// Calls CyclicLogic of every registered CoE transfer and drops the ones that finished.
METHOD PRIVATE ServiceCoeTransfers
VAR
	i : UINT;
END_VAR
i := 0;
WHILE i < ActiveCoeCount DO
	ActiveCoe[i].CyclicLogic();
	IF ActiveCoe[i].Busy THEN
		i := i + 1;
	ELSE
		(* finished: move the last entry into the gap and service it in this cycle as well *)
		ActiveCoeCount			  := ActiveCoeCount - 1;
		ActiveCoe[i]			  := ActiveCoe[ActiveCoeCount];
		ActiveCoe[ActiveCoeCount] := 0;
	END_IF
END_WHILE
END_METHOD

METHOD PROTECTED SetError
VAR_INPUT
	Source	: E_EcErrorSource;
	ErrorId : UDINT;
END_VAR
_Error		 := TRUE;
_ErrorSource := Source;
_ErrorId	 := ErrorId;
END_METHOD

{attribute 'monitoring' := 'call'}
PROPERTY Simulated : BOOL
GET
Simulated := _Simulated;
END_GET
SET
_Simulated := Simulated;
END_SET
END_PROPERTY

{attribute 'monitoring' := 'call'}
PROPERTY SlaveCount : UINT
GET
SlaveCount := EcMaster.SlaveCount;
END_GET
END_PROPERTY

// TRUE if the slave is not in OP with a clean link (any state or link bit set).
METHOD PROTECTED SlaveNeedsDiagnostic : BOOL
VAR_INPUT
	Index : UINT;
END_VAR
SlaveNeedsDiagnostic := (SlavesState[Index].deviceState <> EC_DEVICE_STATE_OP) OR (SlavesState[Index].linkState <> 0);
END_METHOD

// Slave diagnostic sequence, run on every trigger (ChangeCount, slave count, frame WC state):
//  10/11 read all slave states (sized to the configured count)
//  12    classify, SLAVES_PER_CYCLE slaves per cycle; a clean network ends here
//  20/21 read the topology (hot connect flags) - only when a slave needs a diagnostic
//  30    evaluate from the first suspicious slave, stop at the first fault
//  40    assign the sync unit of every slave, once, after the sync units resolved their lists
METHOD PROTECTED SlaveState : BOOL
VAR
	k	: UINT;
	Idx : DINT;
END_VAR
GetSlaveTopologyInfo(sNetId	  := _MasterAmsNetId,
					 pAddrBuf := ADR(SlaveTopologyInfo),
					 cbBufLen := TopologyBufLen(),
					 tTimeout := ADS_TIMEOUT);

GetAllSlaveStates(sNetId	:= _MasterAmsNetId,
				  pStateBuf := ADR(SlavesState),
				  cbBufLen	:= SlaveCountUsed * SIZEOF(SlavesState[0]),
				  tTimeout	:= ADS_TIMEOUT);

CASE SlaveSequence OF
	(* Wait for a trigger *)
	0:
		IF RunSlaveDiag THEN
			RunSlaveDiag  := FALSE;
			SlaveSequence := 10;
		ELSIF NOT SyncUnitsAssigned AND_THEN SyncUnitsResolved() THEN
			EndDiagnosticPass();
		END_IF

	(* Read slave states *)
	10:
		GetAllSlaveStates.bExecute := TRUE;
		WaitCycles				   := 0;
		NextMinorStep(SlaveSequence);

	11:
		IF GetAllSlaveStates.bBusy THEN
			IF AdsWatchdogExpired(ADS_WAIT_CYCLES) THEN
				GetAllSlaveStates.bExecute := FALSE;
				FailSequence(E_EcErrorSource.Ads, ERROR_ADS_TIMEOUT);
			END_IF
		ELSIF GetAllSlaveStates.bError THEN
			GetAllSlaveStates.bExecute := FALSE;
			FailSequence(E_EcErrorSource.Ads, GetAllSlaveStates.nErrId);
		ELSE
			GetAllSlaveStates.bExecute := FALSE;
			ScanIndex				   := 0;
			AnyDiag					   := FALSE;
			FirstDiagIndex			   := 0;
			NextMinorStep(SlaveSequence);
		END_IF

	(* Classify: find the first slave that needs a diagnostic *)
	12:
		FOR k := 1 TO SLAVES_PER_CYCLE DO
			IF ScanIndex >= SlaveCountUsed THEN
				EXIT;
			END_IF

			IF SlaveNeedsDiagnostic(ScanIndex) THEN
				AnyDiag		   := TRUE;
				FirstDiagIndex := ScanIndex;
				EXIT;
			END_IF

			ScanIndex := ScanIndex + 1;
		END_FOR

		IF AnyDiag THEN
			SlaveSequence := 20;
		ELSIF ScanIndex >= SlaveCountUsed THEN
			EndDiagnosticPass(); // every slave OP with a clean link: no topology read, no evaluation
		END_IF

	(* Update topology *)
	20:
		GetSlaveTopologyInfo.bExecute := TRUE;
		WaitCycles					  := 0;
		NextMinorStep(SlaveSequence);

	21:
		IF GetSlaveTopologyInfo.bBusy THEN
			IF AdsWatchdogExpired(ADS_WAIT_CYCLES) THEN
				GetSlaveTopologyInfo.bExecute := FALSE;
				FailSequence(E_EcErrorSource.Ads, ERROR_ADS_TIMEOUT);
			END_IF
		ELSIF GetSlaveTopologyInfo.bError THEN
			GetSlaveTopologyInfo.bExecute := FALSE;
			FailSequence(E_EcErrorSource.Ads, GetSlaveTopologyInfo.nErrId);
		ELSE
			GetSlaveTopologyInfo.bExecute := FALSE;
			ScanIndex					  := FirstDiagIndex;
			SlaveSequence				  := 30;
		END_IF

	(* Evaluate slave errors from the first suspicious slave on *)
	30:
		FOR k := 1 TO SLAVES_PER_CYCLE DO
			IF ScanIndex >= SlaveCountUsed THEN
				EXIT;
			END_IF

			IF EvaluateSlave(ScanIndex) THEN
				ScanIndex := SlaveCountUsed; // fault latched: stop the pass
				EXIT;
			END_IF

			ScanIndex := ScanIndex + 1;
		END_FOR

		IF ScanIndex >= SlaveCountUsed THEN
			EndDiagnosticPass();
		END_IF

	(* Assign the sync unit of every slave (once) *)
	40:
		FOR k := 1 TO SLAVES_PER_CYCLE DO
			IF SyncUnitScan >= SYNC_UNITS THEN
				EXIT;
			END_IF

			IF ScanIndex >= SyncUnit[SyncUnitScan].SlaveCount THEN
				SyncUnitScan := SyncUnitScan + 1;
				ScanIndex	 := 0;
			ELSE
				Idx := GetSlaveIndexByAddr(SyncUnit[SyncUnitScan].SlaveAddress(ScanIndex));
				IF Idx >= 0 THEN
					IoDevice[Idx].SyncUnit := SyncUnit[SyncUnitScan];
				END_IF

				ScanIndex := ScanIndex + 1;
			END_IF
		END_FOR

		IF SyncUnitScan >= SYNC_UNITS THEN
			SyncUnitsAssigned := TRUE;
			SlaveSequence	  := 0;
		END_IF

ELSE
	(* Sequence error: unknown step *)
	FailSequence(E_EcErrorSource.Sequence, SlaveSequence);
END_CASE
END_METHOD

// TRUE once every sync unit has read and resolved its slave list.
METHOD PRIVATE SyncUnitsResolved : BOOL
VAR
	i : UINT;
END_VAR
SyncUnitsResolved := TRUE;
FOR i := 0 TO (SYNC_UNITS - 1) DO
	IF NOT SyncUnit[i].SlavesResolved THEN
		SyncUnitsResolved := FALSE;
		RETURN;
	END_IF
END_FOR
END_METHOD

// Byte length of the topology read: one entry per configured slave, not the whole array.
METHOD PRIVATE TopologyBufLen : UDINT
TopologyBufLen := SlaveCountUsed * SIZEOF(SlaveTopologyInfo[0]);
END_METHOD

END_FUNCTION_BLOCK

// ---- Component/CyclicComponent.TcPOU
FUNCTION_BLOCK ABSTRACT CyclicComponent EXTENDS Component IMPLEMENTS I_Cyclic
VAR
	RegisteredAsCyclicResult : RegistrationResult;
END_VAR

METHOD ABSTRACT CyclicLogic
END_METHOD

METHOD DeregisterWithParent
VAR_INPUT
	Parent : I_ContainComponents;
END_VAR
Parent.DeregisterComponent(THIS^);
Parent.DeregisterCyclic(THIS^);
END_METHOD

METHOD RegisterWithParent
VAR_INPUT
	Parent : I_ContainComponents;
END_VAR
RegisteredAsComponentResult := Parent.RegisterComponent(THIS^);
RegisteredAsCyclicResult := Parent.RegisterCyclic(THIS^);
END_METHOD

END_FUNCTION_BLOCK

// ---- Component/Component.TcPOU
FUNCTION_BLOCK ABSTRACT Component IMPLEMENTS I_Component
VAR
	_Name : T_MaxString;
	RegisteredAsComponentResult : RegistrationResult;
END_VAR

METHOD Accept
VAR_INPUT
	ComponentVisitor : I_ComponentVisitor;
END_VAR
ComponentVisitor.VisitComponent(THIS^);
END_METHOD

METHOD DeregisterWithParent
VAR_INPUT
	Parent : I_ContainComponents;
END_VAR
Parent.DeregisterComponent(THIS^);
END_METHOD

//FB_Init is always available implicitly and it is used primarily for initialization.

//The return value is not evaluated. For a specific influence, you can also declare the

//methods explicitly and provide additional code there with the standard initialization

//code. You can evaluate the return value.
METHOD FB_Init : BOOL
VAR_INPUT
	bInitRetains : BOOL; // TRUE: the retain variables are initialized (reset warm / reset cold)
	bInCopyCode	 : BOOL; // TRUE: the instance will be copied to the copy code afterward (online change)   
	Name		 : T_MaxString;
END_VAR
_Name := Name;
END_METHOD

{attribute 'monitoring' := 'call'}
PROPERTY Name : T_MaxString
GET
Name := _Name;
END_GET
SET
_Name := Name;
END_SET
END_PROPERTY

METHOD RegisterWithParent
VAR_INPUT
	Parent : I_ContainComponents;
END_VAR
RegisteredAsComponentResult := Parent.RegisterComponent(THIS^);
END_METHOD

END_FUNCTION_BLOCK

// ---- Components/EtherCat/SyncUnitTask.TcPOU
{attribute 'no_explicit_call' := 'do not call this POU directly'}
FUNCTION_BLOCK FINAL SyncUnitTask EXTENDS CyclicComponent IMPLEMENTS I_SyncUnitTask, I_Initializable, I_TaskResult, I_Simulatable
VAR
	SyncUnitTaskInfo AT %I* : ST_EtherCatSyncUnitTaskInfo;
	_SlaveCount				: UINT;
	_IsHotConnect			: BOOL;
	_SlavesResolved			: BOOL;
	// Resolves sync unit slave addresses to configured slaves (implemented by EtherCatMaster)
	Registry				: I_EcSlaveRegistry;
	SyncUnitSlaveAddresses	: ARRAY[0..MAX_EC_SLAVES] OF UINT;
	// TRUE at the configured slave index of every slave in this sync unit (filled by the resolve pass)
	MemberByIndex			: ARRAY[0..MAX_EC_SLAVES] OF BOOL;
END_VAR

VAR
	{attribute 'hide'}
	_Initialized : BOOL;
	{attribute 'hide'}
	_Error : BOOL;
	{attribute 'hide'}
	_Busy : BOOL;
	{attribute 'hide'}
	_ErrorId : UDINT;
	{attribute 'hide'}
	_Simulated : BOOL;
END_VAR

VAR
	SyncUnitState			  : UDINT := READ_SLAVES;
	ScanIndex				  : UINT;  // position of the multi-cycle resolve pass
	WaitCycles				  : UDINT; // ADS watchdog and retry delay
	ReadErrorLogged			  : BOOL;
	SlaveMessagePartA		  : STRING;
	SlaveMessagePartB		  : STRING;
	_EventProvider			  : I_EtherCatDiagnosticEventProvider;
	EcGetAllSyncUnitSlaveAddr : FB_EcGetAllSyncUnitSlaveAddr;
END_VAR

VAR CONSTANT
	ERROR_READ_SLAVE_NAMES	   : UDINT := 1;
	ERROR_REGISTER_SYNC_UNIT   : UDINT := 2;
	ERROR_VALID_DATA_SYNC_UNIT : UDINT := 3;
	STRING_LEN				   : INT   := 80;
	SYNC_UNIT_ALARM_MAX		   : UINT  := 3;

	//
	READ_SLAVES			  : UDINT := 0;
	READ_SLAVES_DONE	  : UDINT := 1;
	SYNC_UNIT_OK		  : UDINT := 2;
	RESOLVE_SLAVES		  : UDINT := 3;
	WORKING_COUNTER_ERROR : UDINT := 4;
	READ_ERROR			  : UDINT := 5;
	READ_RETRY_WAIT		  : UDINT := 6;
END_VAR

// Appends the name to the two event message parts while they have room (STRING_LEN each).
METHOD PRIVATE AppendSlaveName
VAR_INPUT
	SlaveName : STRING;
END_VAR

VAR
	Entry : STRING;
END_VAR
IF LEN(SlaveName) = 0 THEN
	RETURN;
END_IF

Entry := CONCAT(SlaveName, ', ');
IF (LEN(Entry) + LEN(SlaveMessagePartA)) <= STRING_LEN THEN
	SlaveMessagePartA := CONCAT(SlaveMessagePartA, Entry);
ELSIF (LEN(Entry) + LEN(SlaveMessagePartB)) <= STRING_LEN THEN
	SlaveMessagePartB := CONCAT(SlaveMessagePartB, Entry);
END_IF
END_METHOD

{attribute 'monitoring' := 'call'}
PROPERTY Busy : BOOL
GET
Busy := _Busy;
END_GET
END_PROPERTY

METHOD PUBLIC CyclicLogic
VAR
	k	 : UINT;
	Addr : UINT;
	Idx	 : DINT;
END_VAR
IF NOT Initialized THEN
	Initialize();
	RETURN;
END_IF

IF Simulated THEN
	RETURN;
END_IF

(* The slave list of a sync unit is configuration data: it is read once (retried on failure) and
   never re-read on working counter recovery. The buffer is sized to the configured slave count. *)
EcGetAllSyncUnitSlaveAddr(sNetId	:= '',
						  nObjectId := SyncUnitTaskInfo.ObjectId,
						  pAddrBuf	:= ADR(SyncUnitSlaveAddresses),
						  cbBufLen	:= SIZEOF(UINT) * MIN(Registry.ConfiguredSlaveCount, MAX_EC_SLAVES + 1),
						  tTimeout	:= T#5S);

EcGetAllSyncUnitSlaveAddr.bExecute := FALSE;
CASE SyncUnitState OF
	READ_SLAVES:
		EcGetAllSyncUnitSlaveAddr.bExecute := TRUE;
		WaitCycles						   := 0;
		SyncUnitState					   := READ_SLAVES_DONE;

	READ_SLAVES_DONE:
		IF EcGetAllSyncUnitSlaveAddr.bBusy THEN
			WaitCycles := WaitCycles + 1;
			IF WaitCycles > ADS_WAIT_CYCLES THEN
				SyncUnitState := READ_ERROR;
			END_IF
		ELSIF EcGetAllSyncUnitSlaveAddr.bError THEN
			SyncUnitState := READ_ERROR;
		ELSE
			_SlaveCount		  := EcGetAllSyncUnitSlaveAddr.nSlaves;
			ScanIndex		  := 0;
			_IsHotConnect	  := FALSE;
			SlaveMessagePartA := '';
			SlaveMessagePartB := '';
			MEMSET(ADR(MemberByIndex), 0, SIZEOF(MemberByIndex));
			SyncUnitState	  := RESOLVE_SLAVES;
		END_IF

	RESOLVE_SLAVES:
		(* Map every address to its configured slave through the slave registry of the master:
		   O(n) in total, SLAVES_PER_CYCLE slaves per cycle. *)
		FOR k := 1 TO SLAVES_PER_CYCLE DO
			IF ScanIndex >= _SlaveCount THEN
				EXIT;
			END_IF

			Addr := SyncUnitSlaveAddresses[ScanIndex];
			IF Addr <> 0 THEN
				Idx := Registry.GetSlaveIndexByAddr(Addr);
				IF Idx >= 0 THEN
					MemberByIndex[Idx] := TRUE;
					_IsHotConnect	   := _IsHotConnect OR Registry.IsHotConnectMember(DINT_TO_UINT(Idx));
					AppendSlaveName(Registry.GetSlaveName(DINT_TO_UINT(Idx)));
				END_IF
			END_IF

			ScanIndex := ScanIndex + 1;
		END_FOR

		IF ScanIndex >= _SlaveCount THEN
			_SlavesResolved := TRUE;
			SyncUnitState	:= SYNC_UNIT_OK;
		END_IF

	SYNC_UNIT_OK:
		IF SyncUnitTaskInfo.WcState THEN
			SyncUnitState := WORKING_COUNTER_ERROR;
			_Busy		  := TRUE;
		ELSE
			_Error	 := FALSE;
			_ErrorID := 0;
			_Busy	 := FALSE;
		END_IF

	WORKING_COUNTER_ERROR:
		_Busy	 := FALSE;
		_Error	 := TRUE;
		_ErrorID := ERROR_VALID_DATA_SYNC_UNIT;
		IF _EventProvider <> 0 THEN
			IF _IsHotConnect THEN
				_EventProvider.RaiseSyncUnitEvent(E_SyncUnit.SyncUnitWarning,
												  _Name,
												  SlaveMessagePartA,
												  SlaveMessagePartB);
			ELSE
				_EventProvider.RaiseSyncUnitEvent(E_SyncUnit.SyncUnitError,
												  _Name,
												  SlaveMessagePartA,
												  SlaveMessagePartB);
			END_IF
		END_IF

		IF NOT SyncUnitTaskInfo.WcState THEN
			IF _EventProvider <> 0 THEN
				_EventProvider.Reset();
			END_IF

			SyncUnitState := SYNC_UNIT_OK; // membership does not change on WC recovery: no re-read
		END_IF

	READ_ERROR:
		IF NOT ReadErrorLogged THEN
			Trace.LogMessage(Name, CONCAT('Sync Unit slave addresses could not be read! Error ID: ', TO_STRING(EcGetAllSyncUnitSlaveAddr.nErrId)));
			ReadErrorLogged := TRUE;
		END_IF

		_Error		  := TRUE;
		_ErrorID	  := ERROR_READ_SLAVE_NAMES;
		WaitCycles	  := 0;
		SyncUnitState := READ_RETRY_WAIT;

	READ_RETRY_WAIT:
		WaitCycles := WaitCycles + 1;
		IF WaitCycles > ADS_WAIT_CYCLES THEN
			SyncUnitState := READ_SLAVES;
		END_IF
END_CASE
END_METHOD

{attribute 'monitoring' := 'call'}
PROPERTY Error : BOOL
GET
Error := _Error;
END_GET
END_PROPERTY

{attribute 'monitoring' := 'call'}
PROPERTY ErrorId : UDINT
GET
ErrorId := _ErrorId;
END_GET
END_PROPERTY

PROPERTY EventProvider : I_EtherCatDiagnosticEventProvider
SET
_EventProvider := EventProvider;
END_SET
END_PROPERTY

(*FB_Init is always available implicitly and it is used primarily for initialization.
The return value is not evaluated. For a specific influence, you can also declare the
methods explicitly and provide additional code there with the standard initialization
code. You can evaluate the return value.*)
METHOD FB_Init : BOOL
VAR_INPUT
	(* TRUE: the retain variables are initialized (reset warm / reset cold)*)
	bInitRetains : BOOL;

	(* TRUE: the instance will be copied to the copy code afterward (online change)   *)
	bInCopyCode			: BOOL;
	Name	 : T_MaxString;
	Registry : I_EcSlaveRegistry;
END_VAR
THIS^.Registry := Registry;
END_METHOD

METHOD Initialize
VAR_INPUT
END_VAR
IF NOT _Error AND NOT Simulated AND F_GetMappingStatus(ADR(SyncUnitTaskInfo.ObjectId), SIZEOF(SyncUnitTaskInfo.ObjectId)) = EplcMappingStatus.MS_Unmapped THEN
	_Error := TRUE;
	Trace.LogMessage(Name, 'Init Failed - SyncUnitTaskInfo.ObjectId not mapped to the sync unit diagnostic!');
END_IF

IF NOT _Error AND NOT Simulated AND F_GetMappingStatus(ADR(SyncUnitTaskInfo.SlaveCount), SIZEOF(SyncUnitTaskInfo.SlaveCount)) = EplcMappingStatus.MS_Unmapped THEN
	_Error := TRUE;
	Trace.LogMessage(Name, 'Init Failed - SyncUnitTaskInfo.SlaveCount not mapped to the sync unit diagnostic!');
END_IF

IF NOT _Error AND NOT Simulated AND F_GetMappingStatus(ADR(SyncUnitTaskInfo.State), SIZEOF(SyncUnitTaskInfo.State)) = EplcMappingStatus.MS_Unmapped THEN
	_Error := TRUE;
	Trace.LogMessage(Name, 'Init Failed - SyncUnitTaskInfo.State not mapped to the sync unit diagnostic!');
END_IF

IF NOT _Error AND NOT Simulated AND F_GetMappingStatus(ADR(SyncUnitTaskInfo.WcState), SIZEOF(SyncUnitTaskInfo.WcState)) = EplcMappingStatus.MS_Unmapped THEN
	_Error := TRUE;
	Trace.LogMessage(Name, 'Init Failed - SyncUnitTaskInfo.WcState not mapped to the sync unit diagnostic!');
END_IF

IF _Error THEN
	RETURN;
END_IF

IF Simulated THEN
	_Initialized := TRUE;
	RETURN;
END_IF

F_EcGetSyncUnitName(SyncUnitTaskInfo.ObjectId, sSyncUnitName => _Name);
_Initialized := TRUE;
END_METHOD

{attribute 'monitoring' := 'call'}
PROPERTY Initialized : BOOL
GET
Initialized := _Initialized;
END_GET
SET
_Initialized := Initialized;
END_SET
END_PROPERTY

{attribute 'monitoring' := 'call'}
PROPERTY IoDataValid : BOOL
GET
IoDataValid := NOT SyncUnitTaskInfo.WcState;
END_GET
END_PROPERTY

// TRUE if at least one slave of this sync unit belongs to a hot connect group.
{attribute 'monitoring' := 'call'}
PROPERTY IsHotConnect : BOOL
GET
IsHotConnect := _IsHotConnect;
END_GET
END_PROPERTY

// O(1) once the slave list is resolved (SlavesResolved).
METHOD IsTerminalPartOfSyncUnit : BOOL
VAR_INPUT
	Addr : UINT;
END_VAR

VAR
	Idx : DINT;
END_VAR
Idx						 := Registry.GetSlaveIndexByAddr(Addr);
IsTerminalPartOfSyncUnit := (Idx >= 0) AND_THEN MemberByIndex[Idx];
END_METHOD

{attribute 'monitoring' := 'call'}
PROPERTY Simulated : BOOL
GET
Simulated := _Simulated;
END_GET
SET
_Simulated := Simulated;
END_SET
END_PROPERTY

// EtherCAT address of the slave at Position (0..SlaveCount-1) in this sync unit; 0 if out of range.
METHOD SlaveAddress : UINT
VAR_INPUT
	Position : UINT;
END_VAR
IF Position < _SlaveCount THEN
	SlaveAddress := SyncUnitSlaveAddresses[Position];
END_IF
END_METHOD

{attribute 'monitoring' := 'call'}
PROPERTY PUBLIC SlaveCount : UINT
GET
SlaveCount := _SlaveCount;
END_GET
END_PROPERTY

// TRUE once the slave list has been read and mapped to the configured slaves.
{attribute 'monitoring' := 'call'}
PROPERTY SlavesResolved : BOOL
GET
SlavesResolved := _SlavesResolved;
END_GET
END_PROPERTY

END_FUNCTION_BLOCK

// ---- Tracing/Trace.TcPOU
FUNCTION_BLOCK Trace
VAR_GENERIC CONSTANT
	MaxCount : UDINT := 10;
END_VAR IMPLEMENTS I_TracePublisher, I_Trace, I_TraceLogger
VAR
	Loggers : ARRAY[0..MaxCount] OF I_TraceLogger;
	_TraceLevel : TcEventSeverityExt := TcEventSeverityExt.Warning;
END_VAR

METHOD Critical
VAR_INPUT
	Source	  : T_MaxString;
	Message	  : T_MaxString;
END_VAR
VAR
	i : UDINT;
END_VAR
FOR i := 0 TO MaxCount DO
	IF Loggers[i] <> 0 AND_THEN _TraceLevel < 5 THEN
		Loggers[i].LogMessage(Source,
							  Message,
							  0,
							  0,
							  1,
							  4);
	END_IF
END_FOR
END_METHOD

METHOD Error
VAR_INPUT
	Source	  : T_MaxString;
	Message	  : T_MaxString;
END_VAR
VAR
	i : UDINT;
END_VAR
FOR i := 0 TO MaxCount DO
	IF Loggers[i] <> 0 AND_THEN _TraceLevel < 4 THEN
		Loggers[i].LogMessage(Source,
							  Message,
							  0,
							  0,
							  1,
							  3);
	END_IF
END_FOR
END_METHOD

METHOD Info
VAR_INPUT
	Source	  : T_MaxString;
	Message	  : T_MaxString;
END_VAR
VAR
	i : UDINT;
END_VAR
FOR i := 0 TO MaxCount DO
	IF Loggers[i] <> 0 AND_THEN _TraceLevel < 2 THEN
		Loggers[i].LogMessage(Source,
							  Message,
							  0,
							  0,
							  1,
							  1);
	END_IF
END_FOR
END_METHOD

METHOD LogMessage
VAR_INPUT
	Key		  : T_MaxString;
	Value	  : T_MaxString;
	SourceId  : UDINT := 0;
	TimeStamp : ULINT := 0;
	MessageId : UDINT := 1;
	Severity  : USINT := 1;
END_VAR

VAR
	i : UDINT;
END_VAR
FOR i := 0 TO MaxCount DO
	IF Loggers[i] <> 0 THEN
		Loggers[i].LogMessage(Key,
							  Value,
							  SourceId,
							  TimeStamp,
							  MessageId,
							  Severity);
	END_IF
END_FOR
END_METHOD

METHOD Subscribe
VAR_INPUT
	Logger : I_TraceLogger;
END_VAR

VAR
	i : UDINT;
END_VAR
FOR i := 0 TO ApplicationBaseParameter.MaxCountInCollections DO
	IF Loggers[i] = 0 THEN
		Loggers[i] := Logger;
		EXIT;
	END_IF
END_FOR
END_METHOD

PROPERTY TraceLevel : TcEventSeverityExt
GET
TraceLevel := _TraceLevel;
END_GET
SET
_TraceLevel := TraceLevel;
END_SET
END_PROPERTY

METHOD Unsubscribe
VAR_INPUT
	Logger : I_TraceLogger;
END_VAR

VAR
	i : UDINT;
END_VAR
FOR i := 0 TO ApplicationBaseParameter.MaxCountInCollections DO
	IF Loggers[i] = Logger THEN
		Loggers[i] := 0;
		EXIT;
	END_IF
END_FOR
END_METHOD

METHOD Verbose
VAR_INPUT
	Source	  : T_MaxString;
	Message	  : T_MaxString;
END_VAR
VAR
	i : UDINT;
END_VAR
FOR i := 0 TO MaxCount DO
	IF Loggers[i] <> 0 AND_THEN _TraceLevel = 0 THEN
		Loggers[i].LogMessage(Source,
							  Message,
							  0,
							  0,
							  1,
							  0);
	END_IF
END_FOR
END_METHOD

METHOD Warning
VAR_INPUT
	Source	  : T_MaxString;
	Message	  : T_MaxString;
END_VAR
VAR
	i : UDINT;
END_VAR
FOR i := 0 TO MaxCount DO
	IF Loggers[i] <> 0 AND_THEN _TraceLevel < 3 THEN
		Loggers[i].LogMessage(Source,
							  Message,
							  0,
							  0,
							  1,
							  2);
	END_IF
END_FOR
END_METHOD

END_FUNCTION_BLOCK

// ---- Statemachine/Generic/State.TcPOU
FUNCTION_BLOCK ABSTRACT State IMPLEMENTS I_State
VAR
	Statemachine  : I_Statemachine;
	SequenceState : UDINT;
END_VAR

METHOD Executing : BOOL
Executing := TRUE;
END_METHOD

//FB_Init is always available implicitly and it is used primarily for initialization.

//The return value is not evaluated. For a specific influence, you can also declare the

//methods explicitly and provide additional code there with the standard initialization

//code. You can evaluate the return value.
METHOD FB_Init : BOOL
VAR_INPUT
	bInitRetains : BOOL; // TRUE: the retain variables are initialized (reset warm / reset cold)
	bInCopyCode	 : BOOL; // TRUE: the instance will be copied to the copy code afterward (online change)  
	State		 : DINT;
	Statemachine : I_Statemachine;
END_VAR
THIS^.Statemachine := Statemachine;
IF THIS^.Statemachine <> 0 THEN
	THIS^.Statemachine.States.AddStateAtIndex(State, THIS^);
END_IF
END_METHOD

METHOD Inactive
SequenceState := 0;
END_METHOD

END_FUNCTION_BLOCK

// ---- Statemachine/Generic/Statemachine.TcPOU
FUNCTION_BLOCK Statemachine
VAR_GENERIC CONSTANT
	InitialState : DINT := 1;
END_VAR
EXTENDS CyclicComponent IMPLEMENTS I_Statemachine
VAR
	StateList	  : StateList<TO_DINT(ApplicationBaseParameter.MaxCountInCollections)>;
	_CurrentState : DINT := InitialState;
	{attribute 'hide'}
	DefaultModeController : ModeControl;
	_Mode				  : I_Mode := DefaultModeController;
END_VAR

METHOD ChangeState
VAR_INPUT
	StateCommand : DINT;
END_VAR
IF StateList.NumberOfStates = 0 THEN
	Trace.LogMessage('Statemachine', 'No states defined!');
	RETURN;
END_IF

_CurrentState := StateCommand;
END_METHOD

{attribute 'monitoring' := 'call'}
PROPERTY CurrentState : DINT
GET
CurrentState := _CurrentState;
END_GET
END_PROPERTY

METHOD CyclicLogic
VAR
	i	  : DINT;
	State : I_State;
END_VAR
IF StateList.NumberOfStates = 0 THEN
	RETURN;
END_IF

FOR i := 0 TO (StateList.NumberOfStates - 1) DO
	State := StateList.GetStateAtIndex(i);
	IF State <> 0 THEN
		IF (i = _CurrentState) THEN
			State.Executing();
		ELSE
			State.Inactive();
		END_IF
	END_IF
END_FOR
END_METHOD

PROPERTY Mode : I_Mode
GET
Mode := _Mode;
END_GET
SET
_Mode := Mode;
END_SET
END_PROPERTY

PROPERTY States : I_StateList
GET
States := StateList;
END_GET
END_PROPERTY

END_FUNCTION_BLOCK

// ---- _Internal/Statemachine/StateList.TcPOU
FUNCTION_BLOCK StateList
VAR_GENERIC CONSTANT
	MaxCount : DINT := 10;
END_VAR IMPLEMENTS I_StateList
VAR
	States : ARRAY[0..MaxCount] OF I_State;
END_VAR

METHOD AddStateAtIndex
VAR_INPUT
	Index : DINT;
	State : I_State;
END_VAR
IF Index > MaxCount THEN
	RETURN;
END_IF

States[Index] := State;
END_METHOD

METHOD GetStateAtIndex : I_State
VAR_INPUT
	Index : DINT;
END_VAR
IF Index > MaxCount THEN
	RETURN;
END_IF

GetStateAtIndex := States[Index];
END_METHOD

PROPERTY NumberOfStates : DINT
GET
NumberOfStates := MaxCount;
END_GET
END_PROPERTY

END_FUNCTION_BLOCK

// ---- Modes/ModeControl.TcPOU
FUNCTION_BLOCK ModeControl IMPLEMENTS I_Mode
VAR
	{attribute 'hide'}
	_CurrentMode : DINT := 1;
END_VAR

METHOD ChangeMode
VAR_INPUT
	RequestedMode : DINT;
END_VAR
IF (RequestedMode >= 1) THEN
	_CurrentMode := RequestedMode;
ELSE
	Trace.LogMessage('Mode Controller', 'Requested Mode is not Defined');
END_IF
END_METHOD

{attribute 'monitoring' := 'call'}
PROPERTY CurrentMode : DINT
GET
CurrentMode := _CurrentMode;
END_GET
END_PROPERTY

END_FUNCTION_BLOCK

// ---- Components/EtherCat/EtherCatIoDevice.TcPOU
FUNCTION_BLOCK EtherCatIoDevice EXTENDS CyclicComponent IMPLEMENTS I_EcIoDevice
VAR
	_Config		  : REFERENCE TO ST_EcSlaveConfigData;
	_State		  : REFERENCE TO ST_EcExtendedSlaveState;
	_SyncUnit	  : I_SyncUnitTask;
	_CoeScheduler : I_CoeTransferScheduler;
	_AmsAddr	  : AMSADDR;
	CoeDevice	  : CoeDevice('CoE Terminal');
	{attribute 'hide'}
	NullCoeDevice : NullCoeDevice('Null Terminal');
END_VAR

PROPERTY AmsNetId : AMSNETID
SET
_AmsAddr.netId := AmsNetId;
END_SET
END_PROPERTY

{attribute 'monitoring' := 'call'}
PROPERTY Bootstrap : BOOL
GET
VAR
	DiagByte : BYTE;
END_VAR
IF __ISVALIDREF(_State) THEN
	DiagByte  := _State.deviceState AND 16#0F;
	Bootstrap := DiagByte = EC_DEVICE_STATE_BOOTSTRAP;
END_IF
END_GET
END_PROPERTY

// CoE access of this slave; NullCoeDevice when the slave has no mailbox (or no configuration yet).
PROPERTY CoE : I_CoeDevice
GET
IF NOT __ISVALIDREF(_Config) OR_ELSE _Config.nMailboxInSize = 0 THEN
	CoE := NullCoeDevice;
ELSE
	CoE := CoeDevice;
END_IF
END_GET
SET
END_SET
END_PROPERTY

// Scheduler that services this slave's CoE transfers (set by EtherCatMaster during Initialize).
// Without one, CyclicLogic must be called each cycle while CoE.Busy.
PROPERTY CoeScheduler : I_CoeTransferScheduler
SET
_CoeScheduler		:= CoeScheduler;
CoeDevice.Scheduler := CoeScheduler;
END_SET
END_PROPERTY

PROPERTY Configuration : REFERENCE TO ST_EcSlaveConfigData
GET
Configuration REF= _Config;
END_GET
SET
_Config REF= Configuration;

(* The CoE mailbox is addressed by the EtherCAT address of the slave. *)
IF __ISVALIDREF(_Config) THEN
	_AmsAddr.port	  := _Config.nAddr;
	CoeDevice.AdsAddr REF= _AmsAddr;
END_IF
END_SET
END_PROPERTY

// Services a CoE transfer in flight when no CoeScheduler is attached. With a scheduler
// (the normal case under EtherCatMaster) this method does nothing.
METHOD CyclicLogic
IF _CoeScheduler <> 0 THEN
	RETURN;
END_IF

IF __ISVALIDREF(_Config) AND_THEN _Config.nMailboxInSize <> 0 AND_THEN CoeDevice.Busy THEN
	CoeDevice.CyclicLogic();
END_IF
END_METHOD

// EC_DEVICE_STATE_ERROR: state machine error in the slave (deviceState bit 4).
{attribute 'monitoring' := 'call'}
PROPERTY DeviceError : BOOL
GET
IF __ISVALIDREF(_State) THEN
	DeviceError := _State.deviceState.4;
END_IF
END_GET
END_PROPERTY

// EC_DEVICE_STATE_DISABLED: slave is disabled in the configuration (deviceState bit 7).
{attribute 'monitoring' := 'call'}
PROPERTY Disabled : BOOL
GET
IF __ISVALIDREF(_State) THEN
	Disabled := _State.deviceState.7;
END_IF
END_GET
END_PROPERTY

{attribute 'monitoring' := 'call'}
PROPERTY Init : BOOL
GET
VAR
	DiagByte : BYTE;
END_VAR
IF __ISVALIDREF(_State) THEN
	DiagByte := _State.deviceState AND 16#0F;
	Init	 := DiagByte = EC_DEVICE_STATE_INIT;
END_IF
END_GET
END_PROPERTY

// EC_DEVICE_STATE_INITCMD_ERROR: error while sending the init commands (deviceState bit 6).
{attribute 'monitoring' := 'call'}
PROPERTY InitCmdError : BOOL
GET
IF __ISVALIDREF(_State) THEN
	InitCmdError := _State.deviceState.6;
END_IF
END_GET
END_PROPERTY

// EC_DEVICE_STATE_INVALID_VPRS: vendor id / product code / revision / serial mismatch (deviceState bit 5).
{attribute 'monitoring' := 'call'}
PROPERTY InvalidVPRS : BOOL
GET
IF __ISVALIDREF(_State) THEN
	InvalidVPRS := _State.deviceState.5;
END_IF
END_GET
END_PROPERTY

{attribute 'monitoring' := 'call'}
PROPERTY IoDataValid : BOOL
GET
IF _SyncUnit <> 0 THEN
	IoDataValid := _SyncUnit.IoDataValid;
ELSE
	IoDataValid := TRUE;
END_IF
END_GET
END_PROPERTY

{attribute 'monitoring' := 'call'}
PROPERTY OP : BOOL
GET
VAR
	DiagByte : BYTE;
END_VAR
IF __ISVALIDREF(_State) THEN
	DiagByte := _State.deviceState AND 16#0F;
	OP		 := DiagByte = EC_DEVICE_STATE_OP;
END_IF
END_GET
END_PROPERTY

{attribute 'monitoring' := 'call'}
PROPERTY PreOp : BOOL
GET
VAR
	DiagByte : BYTE;
END_VAR
IF __ISVALIDREF(_State) THEN
	DiagByte := _State.deviceState AND 16#0F;
	PreOp	 := DiagByte = EC_DEVICE_STATE_PREOP;
END_IF
END_GET
END_PROPERTY

{attribute 'monitoring' := 'call'}
PROPERTY SafeOp : BOOL
GET
VAR
	DiagByte : BYTE;
END_VAR
IF __ISVALIDREF(_State) THEN
	DiagByte := _State.deviceState AND 16#0F;
	SafeOp	 := DiagByte = EC_DEVICE_STATE_SAFEOP;
END_IF
END_GET
END_PROPERTY

PROPERTY State : REFERENCE TO ST_EcExtendedSlaveState
GET
State REF= _State;
END_GET
SET
_State REF= State;
END_SET
END_PROPERTY

PROPERTY SyncUnit : I_SyncUnitTask
SET
_SyncUnit := SyncUnit;
END_SET
END_PROPERTY

END_FUNCTION_BLOCK

// ---- Components/CoE/CoeDevice.TcPOU
FUNCTION_BLOCK CoeDevice EXTENDS CyclicComponent IMPLEMENTS I_CoeDevice, I_CoeTransfer
VAR
	{attribute 'hide'}
	_Error : BOOL;
	{attribute 'hide'}
	_Busy : BOOL;
	{attribute 'hide'}
	_ErrorId : UDINT;
	{attribute 'hide'}
	_ActiveIsWrite : BOOL;
	_AdsAddr   : REFERENCE TO AMSADDR;
	_Scheduler : I_CoeTransferScheduler; // optional: services this device while a transfer is in flight
	CoeRead	   : FB_EcCoESdoReadEx;
	CoeWrite   : FB_EcCoESdoWriteEx;
END_VAR

VAR CONSTANT
	ERROR_NO_ADDRESS : UDINT := 16#70B; // ADS: invalid parameter - AdsAddr reference not set
END_VAR

PROPERTY AdsAddr : REFERENCE TO AMSADDR
GET
AdsAddr REF= _AdsAddr;
END_GET
SET
_AdsAddr REF= AdsAddr;
END_SET
END_PROPERTY

{attribute 'monitoring' := 'call'}
PROPERTY Busy : BOOL
GET
Busy := _Busy;
END_GET
END_PROPERTY

// Services the SDO transfer in flight. Call each cycle while Busy; with a Scheduler set the
// scheduler does this for you.
METHOD CyclicLogic
VAR_INST
END_VAR
IF NOT __ISVALIDREF(_AdsAddr) THEN
	RETURN;
END_IF

CoeRead(sNetId := F_CreateAmsNetId(_AdsAddr.netId), nSlaveAddr := _AdsAddr.port, tTimeout := T#1S);
CoeWrite(sNetId := F_CreateAmsNetId(_AdsAddr.netId), nSlaveAddr := _AdsAddr.port, tTimeout := T#1S);
CoeRead.bExecute  := FALSE;
CoeWrite.bExecute := FALSE;

(* Only the active function block decides Busy/Error: a stale bError of the other one must not leak. *)
IF _ActiveIsWrite THEN
	_Busy := CoeWrite.bBusy;
	IF CoeWrite.bError THEN
		_Error	 := TRUE;
		_ErrorId := CoeWrite.nErrId;
	END_IF
ELSE
	_Busy := CoeRead.bBusy;
	IF CoeRead.bError THEN
		_Error	 := TRUE;
		_ErrorId := CoeRead.nErrId;
	END_IF
END_IF
END_METHOD

{attribute 'monitoring' := 'call'}
PROPERTY Error : BOOL
GET
Error := _Error;
END_GET
END_PROPERTY

{attribute 'monitoring' := 'call'}
PROPERTY ErrorId : UDINT
GET
ErrorID := _ErrorID;
END_GET
END_PROPERTY

// Starts an SDO read; ignored while Busy. Fails with ERROR_NO_ADDRESS if AdsAddr is not set.
METHOD Read
VAR_INPUT
	Index	 : WORD;
	SubIndex : BYTE;
	pDstBuf	 : PVOID;
	BufLen	 : UDINT;
END_VAR
IF _Busy THEN
	RETURN;
END_IF

IF NOT __ISVALIDREF(_AdsAddr) THEN
	_Error	 := TRUE;
	_ErrorId := ERROR_NO_ADDRESS;
	RETURN;
END_IF

CoeRead.nSubIndex		:= SubIndex;
CoeRead.nIndex			:= Index;
CoeRead.pDstBuf			:= pDstBuf;
CoeRead.cbBufLen		:= BufLen;
CoeRead.bCompleteAccess := SubIndex = 0;
_ActiveIsWrite			:= FALSE;
_Error					:= FALSE;
_ErrorId				:= 0;
_Busy					:= TRUE;
CoeRead.bExecute		:= TRUE;

IF _Scheduler <> 0 THEN
	_Scheduler.Register(THIS^);
END_IF
END_METHOD

// Optional scheduler that calls CyclicLogic while a transfer is in flight (set by EtherCatIoDevice).
PROPERTY Scheduler : I_CoeTransferScheduler
GET
Scheduler := _Scheduler;
END_GET
SET
_Scheduler := Scheduler;
END_SET
END_PROPERTY

// Starts an SDO write from pDstBuf (used as the source buffer); ignored while Busy.
METHOD Write
VAR_INPUT
	Index	 : WORD;
	SubIndex : BYTE;
	pDstBuf	 : PVOID;
	BufLen	 : UDINT;
END_VAR
IF _Busy THEN
	RETURN;
END_IF

IF NOT __ISVALIDREF(_AdsAddr) THEN
	_Error	 := TRUE;
	_ErrorId := ERROR_NO_ADDRESS;
	RETURN;
END_IF

CoeWrite.nSubIndex		 := SubIndex;
CoeWrite.nIndex			 := Index;
CoeWrite.pSrcBuf		 := pDstBuf;
CoeWrite.cbBufLen		 := BufLen;
CoeWrite.bCompleteAccess := SubIndex = 0;
_ActiveIsWrite			 := TRUE;
_Error					 := FALSE;
_ErrorId				 := 0;
_Busy					 := TRUE;
CoeWrite.bExecute		 := TRUE;

IF _Scheduler <> 0 THEN
	_Scheduler.Register(THIS^);
END_IF
END_METHOD

END_FUNCTION_BLOCK

// ---- Components/CoE/NullCoeDevice.TcPOU
FUNCTION_BLOCK NullCoeDevice EXTENDS CyclicComponent IMPLEMENTS I_CoeDevice
VAR
END_VAR

PROPERTY AdsAddr : REFERENCE TO AMSADDR
GET
END_GET
SET
END_SET
END_PROPERTY

{attribute 'monitoring' := 'call'}
PROPERTY Busy : BOOL
GET
END_GET
END_PROPERTY

METHOD CyclicLogic
END_METHOD

{attribute 'monitoring' := 'call'}
PROPERTY Error : BOOL
GET
END_GET
END_PROPERTY

{attribute 'monitoring' := 'call'}
PROPERTY ErrorId : UDINT
GET
END_GET
END_PROPERTY

METHOD Read
VAR_INPUT
	Index	 : WORD;
	SubIndex : BYTE;
	pDstBuf	 : PVOID;
	BufLen	 : UDINT;
END_VAR
END_METHOD

METHOD Write
VAR_INPUT
	Index	 : WORD;
	SubIndex : BYTE;
	pDstBuf	 : PVOID;
	BufLen	 : UDINT;
END_VAR
END_METHOD

END_FUNCTION_BLOCK

// ---- Motion/MC3/Mc3Axis.TcPOU
FUNCTION_BLOCK Mc3Axis EXTENDS CyclicComponent IMPLEMENTS I_Initializable, I_Mc3Axis
VAR
	_Axis				 : REFERENCE TO Tc3_Mc3Ptp.AXIS_REF;
	Defaults			 : ST_Mc3MotionDefaults;
	MotionTaskCollection : Mc3MotionTaskCollection<ApplicationBaseMotionParameter.MaxMotionTasks>(THIS^);

	// Tasks
	PowerTask  : Mc3PowerTask	 := (Name := 'MC Power');
	JogTask	   : Mc3MoveJogTask	 := (Name := 'MC Jog');
	_StopTask  : I_Mc3MotionTask := Defaults.DefaultStopTask;
	_ResetTask : I_Mc3MotionTask := Defaults.DefaultResetTask;
	_HomeTask  : I_Mc3MotionTask := Defaults.DefaultHomeTask;
	SetOverride : Tc3_Mc3Ptp.MC_SetOverride;

	// Initialization is delegated to its own component
	ParameterLoader : Mc3AxisParameterLoader<ApplicationBaseMotionParameter.MaxAxisParameters>;
	_Initialized		: BOOL;
	// TRUE once a parent module owns our Initialize() call
	{attribute 'hide'}
	_InitializeDrivenByParent : BOOL;
	{attribute 'hide'}
	_LoadErrorLogged		  : BOOL;

	//
	_Acceleration : LREAL;
	_Deceleration : LREAL;
	_Velocity	  : LREAL;
	_Jerk		  : LREAL;
	_McBufferMode : Tc3_Mc3Ptp.EBufferMode		:= Tc3_Mc3Ptp.EBufferMode.Aborting;
	_Direction	  : Tc3_Mc3Ptp.EModuloDirection := Tc3_Mc3Ptp.EModuloDirection.ShortestDistance;
	_JogMode	  : Tc3_Mc3Ptp.EJogMode			:= Tc3_Mc3Ptp.EJogMode.StandardSlow;
END_VAR

{attribute 'monitoring' := 'call'}
PROPERTY Acceleration : LREAL
GET
Acceleration := _Acceleration;
END_GET
SET
_Acceleration := Acceleration;
END_SET
END_PROPERTY

{attribute 'monitoring' := 'call'}
PROPERTY ActualAcceleration : LREAL
GET
ActualAcceleration := _Axis.McToPlc.Act.Acceleration;
END_GET
END_PROPERTY

{attribute 'monitoring' := 'call'}
PROPERTY ActualPosition : LREAL
GET
ActualPosition := _Axis.McToPlc.Act.Position;
END_GET
END_PROPERTY

{attribute 'monitoring' := 'call'}
PROPERTY ActualPositionModulo : LREAL
GET
ActualPositionModulo := _Axis.McToPlc.Modulo.ActPosition;
END_GET
END_PROPERTY

{attribute 'monitoring' := 'call'}
PROPERTY ActualTorque : LREAL
GET
ActualTorque := _Axis.McToPlc.Act.Torque;
END_GET
END_PROPERTY

{attribute 'monitoring' := 'call'}
PROPERTY ActualVelocity : LREAL
GET
ActualVelocity := _Axis.McToPlc.Act.Velocity;
END_GET
END_PROPERTY

PROPERTY Axis : REFERENCE TO Tc3_Mc3Ptp.AXIS_REF
GET
Axis REF= _Axis;
END_GET
END_PROPERTY

PROPERTY BufferMode : REFERENCE TO Tc3_Mc3Ptp.EBufferMode
GET
BufferMode REF= _McBufferMode;
END_GET
END_PROPERTY

{attribute 'monitoring' := 'call'}
PROPERTY Busy : BOOL
GET
Busy := MotionTaskCollection.Busy;
END_GET
END_PROPERTY

METHOD CyclicLogic
IF NOT _Initialized THEN
	// A parent module drives Initialize() through its Initializer. Only
	// self-initialize when there is no parent, so the call has one owner.
	IF NOT _InitializeDrivenByParent THEN
		Initialize();
	END_IF

	RETURN;
END_IF

MotionTaskCollection.CyclicLogic();
END_METHOD

{attribute 'monitoring' := 'call'}
PROPERTY Coupled : BOOL
GET
Coupled := _Axis.McToPlc.Std.AxisState = EAxisState.SynchronizedMotion;
END_GET
END_PROPERTY

{attribute 'monitoring' := 'call'}
PROPERTY Deceleration : LREAL
GET
Deceleration := _Deceleration;
END_GET
SET
_Deceleration := Deceleration;
END_SET
END_PROPERTY

PROPERTY Direction : REFERENCE TO Tc3_Mc3Ptp.EModuloDirection
GET
Direction REF= _Direction;
END_GET
END_PROPERTY

{attribute 'monitoring' := 'call'}
PROPERTY Disabled : BOOL
GET
Disabled := NOT PowerTask.Enabled;
END_GET
END_PROPERTY

METHOD Disable
PowerTask.Disable();
END_METHOD

METHOD Enable
IF Error THEN
	RETURN;
END_IF

PowerTask.Enable();
END_METHOD

{attribute 'monitoring' := 'call'}
PROPERTY Enabled : BOOL
GET
Enabled := PowerTask.Enabled;
END_GET
END_PROPERTY

{attribute 'monitoring' := 'call'}
PROPERTY Error : BOOL
GET
Error := MotionTaskCollection.Error OR (_Axis.McToPlc.Std.AxisState = EAxisState.ErrorStop);
END_GET
END_PROPERTY

{attribute 'monitoring' := 'call'}
PROPERTY ErrorId : UDINT
GET
IF _Axis.McToPlc.Std.ErrorId <> 0 THEN
	ErrorId := _Axis.McToPlc.Std.ErrorId;
	RETURN;
END_IF

ErrorId := MotionTaskCollection.ErrorId;
END_GET
END_PROPERTY

(*FB_Init is always available implicitly and it is used primarily for initialization.
The return value is not evaluated. For a specific influence, you can also declare the
methods explicitly and provide additional code there with the standard initialization
code. You can evaluate the return value.*)
METHOD FB_Init : BOOL
VAR_INPUT
	(* TRUE: the retain variables are initialized (reset warm / reset cold)*)
	bInitRetains : BOOL;

	(* TRUE: the instance will be copied to the copy code afterward (online change)   *)
	bInCopyCode : BOOL;
	Name		: T_MaxString;
	Axis		: REFERENCE TO Tc3_Mc3Ptp.AXIS_REF;
END_VAR
_Axis REF= Axis;

// Declare which NC parameters pre-load the dynamics properties.
// Adding one is a single line here - there is no sequence to edit.
ParameterLoader.Configure(_Axis);
ParameterLoader.AddParameter(EAxisParameterId.DefaultAcceleration, ADR(_Acceleration));
ParameterLoader.AddParameter(EAxisParameterId.DefaultDeceleration, ADR(_Deceleration));
ParameterLoader.AddParameter(EAxisParameterId.DefaultJerk, ADR(_Jerk));
ParameterLoader.AddParameter(EAxisParameterId.MaximumVelocity, ADR(_Velocity));

// Register all Motion Tasks to Collection
MotionTaskCollection.AddTask(PowerTask);
MotionTaskCollection.AddTask(_StopTask);
MotionTaskCollection.AddTask(_ResetTask);
MotionTaskCollection.AddTask(_HomeTask);
MotionTaskCollection.AddTask(JogTask);
END_METHOD

METHOD Home
VAR_INPUT
END_VAR
IF Coupled THEN
	// Homing a coupled axis is meaningless - decouple first
	RETURN;
END_IF

_HomeTask.Execute();
END_METHOD

PROPERTY HomeTask : I_Mc3MotionTask
SET
MotionTaskCollection.RemoveTaskByInstance(_HomeTask);
_HomeTask := HomeTask;
MotionTaskCollection.AddTask(_HomeTask);
END_SET
END_PROPERTY

{attribute 'monitoring' := 'call'}
PROPERTY InhibitFeedBackward : BOOL
GET
InhibitFeedBackward := PowerTask.InhibitFeedBackward;
END_GET
SET
PowerTask.InhibitFeedBackward := InhibitFeedBackward;
END_SET
END_PROPERTY

{attribute 'monitoring' := 'call'}
PROPERTY InhibitFeedForward : BOOL
GET
InhibitFeedForward := PowerTask.InhibitFeedForward;
END_GET
SET
PowerTask.InhibitFeedForward := InhibitFeedForward;
END_SET
END_PROPERTY

METHOD Initialize
IF _Initialized THEN
	RETURN;
END_IF

ParameterLoader.Initialize();

IF ParameterLoader.Initialized THEN
	Trace.LogMessage(_Name, 'Axis initialization complete');
	_Initialized := TRUE;
	RETURN;
END_IF

IF ParameterLoader.Error AND NOT _LoadErrorLogged THEN
	_LoadErrorLogged := TRUE;
	Trace.LogMessage(_Name, 'Axis not initialized - error reading parameter - check links!');
END_IF
END_METHOD

{attribute 'monitoring' := 'call'}
PROPERTY Initialized : BOOL
GET
Initialized := _Initialized;
END_GET
SET
_Initialized := Initialized;
END_SET
END_PROPERTY

{attribute 'monitoring' := 'call'}
PROPERTY Jerk : LREAL
GET
Jerk := _Jerk;
END_GET
SET
_Jerk := Jerk;
END_SET
END_PROPERTY

METHOD Jog
VAR_INPUT
	JogForward	 : BOOL;
	JogBackwards : BOOL;
	Distance	 : LREAL := 0;
END_VAR
IF Error OR Coupled THEN
	RETURN;
END_IF

JogTask.JogBackwards := JogBackwards;
JogTask.JogForward	 := JogForward;
JogTask.Distance	 := Distance;
JogTask.Mode		 := _JogMode;
JogTask.Execute();
END_METHOD

{attribute 'monitoring' := 'call'}
PROPERTY JogMode : E_AxisJogMode
GET
IF _JogMode = Tc3_Mc3Ptp.EJogMode.StandardFast THEN
	JogMode := E_AxisJogMode.Fast;
ELSE
	JogMode := E_AxisJogMode.Slow;
END_IF
END_GET
SET
IF JogMode = E_AxisJogMode.Fast THEN
	_JogMode := Tc3_Mc3Ptp.EJogMode.StandardFast;
ELSE
	_JogMode := Tc3_Mc3Ptp.EJogMode.StandardSlow;
END_IF
END_SET
END_PROPERTY

PROPERTY MotionTasks : I_MotionTaskCollection
GET
MotionTasks := MotionTaskCollection;
END_GET
END_PROPERTY

{attribute 'monitoring' := 'call'}
PROPERTY Override : LREAL // 0-100%
SET
SetOverride(Axis		   := _Axis,
			Enable		   := TRUE,
			VelocityFactor := (Override / 100.0),
			Enabled		   =>,
			Error		   =>,
			ErrorId		   =>);
END_SET
END_PROPERTY

{attribute 'monitoring' := 'call'}
PROPERTY PositionLag : LREAL
GET
PositionLag := _Axis.McToPlc.Act.PositionLag;
END_GET
END_PROPERTY

METHOD RegisterWithParent
VAR_INPUT
	Parent : I_ContainComponents;
END_VAR
SUPER^.RegisterWithParent(Parent);
Parent.RegisterInitialize(THIS^);
_InitializeDrivenByParent := TRUE;
END_METHOD

METHOD Reset
IF _ResetTask.Execute() THEN
	MotionTaskCollection.Reset();
END_IF
END_METHOD

PROPERTY ResetTask : I_Mc3MotionTask
SET
MotionTaskCollection.RemoveTaskByInstance(_ResetTask);
_ResetTask := ResetTask;
MotionTaskCollection.AddTask(_ResetTask);
END_SET
END_PROPERTY

{attribute 'monitoring' := 'call'}
PROPERTY SetAcceleration : LREAL
GET
SetAcceleration := _Axis.McToPlc.Set.Acceleration;
END_GET
END_PROPERTY

{attribute 'monitoring' := 'call'}
PROPERTY SetPosition : LREAL
GET
SetPosition := _Axis.McToPlc.Set.Position;
END_GET
END_PROPERTY

{attribute 'monitoring' := 'call'}
PROPERTY SetPositionModulo : LREAL
GET
SetPositionModulo := _Axis.McToPlc.Modulo.SetPosition;
END_GET
END_PROPERTY

{attribute 'monitoring' := 'call'}
PROPERTY SetVelocity : LREAL
GET
SetVelocity := _Axis.McToPlc.Set.Velocity;
END_GET
END_PROPERTY

METHOD Stop
IF Error AND _Axis.McToPlc.Std.HasError THEN
	(* It's possible that a function block errored but
	not the NC itself--in this case we can allow a stop command.
	If the NC Axis has a real fault then we want a successful reset first *)
	RETURN;
END_IF

_StopTask.Execute();
END_METHOD

{attribute 'monitoring' := 'call'}
PROPERTY Stopped : BOOL
GET
Stopped := (_Axis.McToPlc.Std.AxisState <= EAxisState.Standstill) OR ((_Axis.McToPlc.Std.AxisState = EAxisState.SynchronizedMotion) AND (SetVelocity = 0.0));
END_GET
END_PROPERTY

PROPERTY StopTask : I_Mc3MotionTask
SET
MotionTaskCollection.RemoveTaskByInstance(_StopTask);
_StopTask := StopTask;
MotionTaskCollection.AddTask(_ResetTask);
END_SET
END_PROPERTY

{attribute 'monitoring' := 'call'}
PROPERTY SynchronizedMotion : BOOL
GET
SynchronizedMotion := _Axis.McToPlc.Std.AxisState = EAxisState.SynchronizedMotion;
END_GET
END_PROPERTY

{attribute 'monitoring' := 'call'}
PROPERTY Velocity : LREAL
GET
Velocity := _Velocity;
END_GET
SET
_Velocity := Velocity;
END_SET
END_PROPERTY

END_FUNCTION_BLOCK

// ---- _Internal/MotionTasks/MC3/Base/Mc3MotionTaskCollection.TcPOU
FUNCTION_BLOCK Mc3MotionTaskCollection
VAR_GENERIC CONSTANT
	MaxCount : UDINT := 10;
END_VAR IMPLEMENTS I_Mc3MotionTaskCollection, I_Cyclic, I_Resettable
VAR
	MotionTasks		   : ARRAY[0..MaxCount] OF I_Mc3MotionTask;
	Axis			   : I_Mc3Axis;
	LastBusyTaskState  : ST_TaskState;
	LastErrorTaskState : ST_TaskState;
	CurrentTaskStates  : ARRAY[0..MaxCount] OF ST_TaskState;
	{attribute 'hide'}
	_Busy : BOOL;
	{attribute 'hide'}
	_Error : BOOL;
	{attribute 'hide'}
	_ErrorId : UDINT;
	{attribute 'hide'}
	_ErrorTask : T_MaxString;
END_VAR

METHOD AddTask
VAR_INPUT
	Task : I_Mc3MotionTask;
END_VAR

VAR
	i : UDINT;
END_VAR
Task.Axis := Axis;
FOR i := 0 TO MaxCount DO
	IF MotionTasks[i] = 0 THEN
		MotionTasks[i] := Task;
		EXIT;
	END_IF
END_FOR
END_METHOD

{attribute 'monitoring' := 'call'}
PROPERTY Busy : BOOL
GET
Busy := _Busy;
END_GET
END_PROPERTY

METHOD CyclicLogic
VAR
	MotionTask : I_Mc2MotionTask;
END_VAR

VAR_INST
	i				: UDINT;
END_VAR
_Busy := FALSE;
FOR i := 0 TO MaxCount DO
	IF MotionTasks[i] = 0 THEN
		EXIT;
	END_IF

	MotionTasks[i].CyclicLogic();
	IF MotionTasks[i].Busy THEN
		LastBusyTaskState.Name	  := MotionTasks[i].Name;
		LastBusyTaskState.Busy	  := MotionTasks[i].Busy;
		LastBusyTaskState.Error	  := MotionTasks[i].Error;
		LastBusyTaskState.ErrorId := MotionTasks[i].ErrorId;
		_Busy					  := TRUE;
	END_IF

	IF MotionTasks[i].Error AND NOT _Error THEN
		LastErrorTaskState.Name	   := MotionTasks[i].Name;
		LastErrorTaskState.Busy	   := MotionTasks[i].Busy;
		LastErrorTaskState.Error   := MotionTasks[i].Error;
		LastErrorTaskState.ErrorId := MotionTasks[i].ErrorId;
		_Error					   := TRUE;
		_ErrorId				   := MotionTasks[i].ErrorId;
		_ErrorTask				   := MotionTasks[i].Name;
	END_IF

	CurrentTaskStates[i].Name	 := MotionTasks[i].Name;
	CurrentTaskStates[i].Busy	 := MotionTasks[i].Busy;
	CurrentTaskStates[i].Error	 := MotionTasks[i].Error;
	CurrentTaskStates[i].ErrorId := MotionTasks[i].ErrorId;
END_FOR
END_METHOD

{attribute 'monitoring' := 'call'}
PROPERTY Error : BOOL
GET
Error := _Error;
END_GET
END_PROPERTY

{attribute 'monitoring' := 'call'}
PROPERTY ErrorId : UDINT
GET
ErrorId := _ErrorId;
END_GET
END_PROPERTY

{attribute 'monitoring' := 'call'}
PROPERTY ErrorTask : T_MaxString
GET
ErrorTask := _ErrorTask;
END_GET
END_PROPERTY

//FB_Init is always available implicitly and it is used primarily for initialization.

//The return value is not evaluated. For a specific influence, you can also declare the

//methods explicitly and provide additional code there with the standard initialization

//code. You can evaluate the return value.
METHOD FB_Init : BOOL
VAR_INPUT
	bInitRetains : BOOL; // TRUE: the retain variables are initialized (reset warm / reset cold)
	bInCopyCode	 : BOOL; // TRUE: the instance will be copied to the copy code afterward (online change)  
	Axis		 : I_Mc3Axis;
END_VAR
THIS^.Axis := Axis;
END_METHOD

METHOD RemoveTaskByInstance
VAR_INPUT
	Task : I_Mc3MotionTask;
END_VAR

VAR
	i : UDINT;
END_VAR
FOR i := 0 TO MaxCount DO
	IF MotionTasks[i] = Task THEN
		MotionTasks[i] := 0;
		EXIT;
	END_IF
END_FOR
END_METHOD

METHOD Reset
_Error	   := FALSE;
_ErrorId   := 0;
_ErrorTask := '';
END_METHOD

END_FUNCTION_BLOCK

// ---- _Internal/MotionTasks/MC3/Power/Mc3PowerTask.TcPOU
FUNCTION_BLOCK Mc3PowerTask EXTENDS Mc3MotionTask IMPLEMENTS I_Mc3MotionPowerTask
VAR
	McPower : Tc3_Mc3Ptp.MC_Power;
	{attribute 'hide'}
	_InhibitFeedForward : BOOL;
	{attribute 'hide'}
	_InhibitFeedBackward : BOOL;
END_VAR

{attribute 'monitoring' := 'call'}
PROPERTY Busy : BOOL
GET
Busy := FALSE; (*MC Power Busy behaves busy as long as enabled*)
END_GET
END_PROPERTY

METHOD CyclicLogic
McPower(Axis		   := _Axis.Axis,
		EnablePositive := NOT _InhibitFeedForward,
		EnableNegative := NOT _InhibitFeedBackward,
		Status		   =>,
		Error		   =>,
		ErrorId		   =>);
END_METHOD

METHOD Disable
McPower(Axis		   := _Axis.Axis,
		Enable		   := FALSE,
		EnablePositive := NOT _InhibitFeedForward,
		EnableNegative := NOT _InhibitFeedBackward,
		Status		   =>,
		Error		   =>,
		ErrorId		   =>);
END_METHOD

METHOD Enable
McPower(Axis		   := _Axis.Axis,
		Enable		   := TRUE,
		EnablePositive := NOT _InhibitFeedForward,
		EnableNegative := NOT _InhibitFeedBackward,
		Status		   =>,
		Error		   =>,
		ErrorId		   =>);
END_METHOD

{attribute 'monitoring' := 'call'}
PROPERTY Enabled : BOOL
GET
Enabled := McPower.Status;
END_GET
END_PROPERTY

{attribute 'monitoring' := 'call'}
PROPERTY Error : BOOL
GET
Error := McPower.Error;
END_GET
END_PROPERTY

{attribute 'monitoring' := 'call'}
PROPERTY ErrorId : UDINT
GET
ErrorId := McPower.ErrorID;
END_GET
END_PROPERTY

METHOD Execute : BOOL
Execute := TRUE;
END_METHOD

{attribute 'monitoring' := 'call'}
PROPERTY InhibitFeedBackward : BOOL
GET
InhibitFeedBackward := _InhibitFeedBackward;
END_GET
SET
_InhibitFeedBackward := InhibitFeedBackward;
END_SET
END_PROPERTY

{attribute 'monitoring' := 'call'}
PROPERTY InhibitFeedForward : BOOL
GET
InhibitFeedForward := _InhibitFeedForward;
END_GET
SET
_InhibitFeedForward := InhibitFeedForward;
END_SET
END_PROPERTY

END_FUNCTION_BLOCK

// ---- _Internal/MotionTasks/MC3/Base/Mc3MotionTask.TcPOU
FUNCTION_BLOCK ABSTRACT Mc3MotionTask IMPLEMENTS I_Mc3MotionTask
VAR
	_Name : T_MaxString;
	_Axis : I_Mc3Axis;
END_VAR

PROPERTY Axis : I_Mc3Axis
GET
Axis := _Axis;
END_GET
SET
_Axis := Axis;
END_SET
END_PROPERTY

{attribute 'monitoring' := 'call'}
PROPERTY ABSTRACT Busy : BOOL
GET
END_GET
END_PROPERTY

METHOD ABSTRACT CyclicLogic
END_METHOD

{attribute 'monitoring' := 'call'}
PROPERTY ABSTRACT Error : BOOL
GET
END_GET
END_PROPERTY

{attribute 'monitoring' := 'call'}
PROPERTY ABSTRACT ErrorId : UDINT
GET
END_GET
END_PROPERTY

METHOD ABSTRACT Execute : BOOL;
END_METHOD

{attribute 'monitoring' := 'call'}
PROPERTY Name : T_MaxString
GET
Name := _Name;
END_GET
SET
_Name := Name;
END_SET
END_PROPERTY

END_FUNCTION_BLOCK

// ---- _Internal/MotionTasks/MC3/Move/Mc3MoveJogTask.TcPOU
FUNCTION_BLOCK Mc3MoveJogTask EXTENDS Mc3MotionTask IMPLEMENTS I_Mc3MotionJogTask
VAR
	McJog		  : Tc3_Mc3Ptp.MC_Jog;
	_JogForward	  : BOOL;
	_JogBackwards : BOOL;
	_Mode		  : Tc3_Mc3Ptp.EJogMode;
	_Distance	  : LREAL;
END_VAR

{attribute 'monitoring' := 'call'}
PROPERTY Busy : BOOL
GET
Busy := MCJog.Busy;
END_GET
END_PROPERTY

METHOD CyclicLogic
IF McJog.Error OR _Axis.Error THEN
	_JogForward	  := FALSE;
	_JogBackwards := FALSE;
END_IF

McJog(Axis			 := _Axis.Axis,
	  JogForward	 := _JogForward,
	  JogBackward	 := _JogBackwards,
	  Mode			 := _Mode,
	  Distance		 := _Distance,
	  Velocity		 := _Axis.Velocity,
	  Acceleration	 := _Axis.Acceleration,
	  Deceleration	 := _Axis.Deceleration,
	  Jerk			 := _Axis.Jerk,
	  Done			 =>,
	  Busy			 =>,
	  Active		 =>,
	  CommandAborted =>,
	  Error			 =>,
	  ErrorId		 =>);
END_METHOD

PROPERTY Distance : LREAL
SET
_Distance:= Distance;
END_SET
END_PROPERTY

{attribute 'monitoring' := 'call'}
PROPERTY Error : BOOL
GET
Error := MCJog.Error;
END_GET
END_PROPERTY

{attribute 'monitoring' := 'call'}
PROPERTY ErrorId : UDINT
GET
ErrorId := MCJog.ErrorID;
END_GET
END_PROPERTY

METHOD Execute : BOOL
McJog(Axis			 := _Axis.Axis,
	  JogForward	 := _JogForward,
	  JogBackward	 := _JogBackwards,
	  Mode			 := _Mode,
	  Distance		 := _Distance,
	  Velocity		 := _Axis.Velocity,
	  Acceleration	 := _Axis.Acceleration,
	  Deceleration	 := _Axis.Deceleration,
	  Jerk			 := _Axis.Jerk,
	  Done			 =>,
	  Busy			 =>,
	  Active		 =>,
	  CommandAborted =>,
	  Error			 =>,
	  ErrorId		 =>);
END_METHOD

PROPERTY JogBackwards : BOOL
SET
_JogBackwards := JogBackwards;
END_SET
END_PROPERTY

PROPERTY JogForward : BOOL
SET
_JogForward := JogForward;
END_SET
END_PROPERTY

PROPERTY Mode : Tc3_Mc3Ptp.EJogMode
SET
_Mode := Mode;
END_SET
END_PROPERTY

END_FUNCTION_BLOCK

// ---- Motion/MC3/Mc3AxisParameterLoader.TcPOU
(* Reads a table of NC axis parameters into the owning axis, one parameter per
   MC_ReadParameter call, and reports completion through I_Initializable.

   Adding a parameter is a single AddParameter() call at construction time -
   there is no sequence to edit. Call Configure() once with the axis reference,
   then AddParameter() for each value, then Initialize() cyclically until
   Initialized or Error. *)
FUNCTION_BLOCK Mc3AxisParameterLoader
VAR_GENERIC CONSTANT
	MaxParameters : UDINT := 10;
END_VAR IMPLEMENTS I_Initializable
VAR
	_Axis		  : REFERENCE TO Tc3_Mc3Ptp.AXIS_REF;
	_Bindings	  : ARRAY[1..MaxParameters] OF ST_Mc3ParameterBinding;
	_Count		  : UDINT;
	_Index		  : UDINT := 1;
	_Initialized  : BOOL;
	_Error		  : BOOL;
	_ErrorId	  : UDINT;
	_Overflow	  : BOOL;
	_Value		  : LREAL;
	ReadParameter : Tc3_Mc3Ptp.MC_ReadParameter;
END_VAR

(* Registers one parameter to be read into Target.
   Idempotent: re-registering a ParameterId updates its Target rather than
   adding a second entry, so an online change re-running FB_Init refreshes the
   pointers instead of growing the table.
   Returns FALSE when the table is full or Target is invalid. *)
METHOD AddParameter : BOOL
VAR_INPUT
	ParameterId : Tc3_Mc3Ptp.EAxisParameterId;
	Target		: POINTER TO LREAL;
END_VAR

VAR
	i : UDINT;
END_VAR
IF Target = 0 THEN
	RETURN;
END_IF

// Already registered - just refresh the target pointer
FOR i := 1 TO _Count DO
	IF _Bindings[i].ParameterId = ParameterId THEN
		_Bindings[i].Target := Target;
		AddParameter		:= TRUE;
		RETURN;
	END_IF
END_FOR

IF _Count >= MaxParameters THEN
	_Overflow := TRUE;
	RETURN;
END_IF

_Count := _Count + 1;
_Bindings[_Count].ParameterId := ParameterId;
_Bindings[_Count].Target	  := Target;
AddParameter := TRUE;
END_METHOD

(* Binds the loader to the NC axis it should read from. *)
METHOD Configure
VAR_INPUT
	Axis : REFERENCE TO Tc3_Mc3Ptp.AXIS_REF;
END_VAR
_Axis REF= Axis;
END_METHOD

{attribute 'monitoring' := 'call'}
PROPERTY Error : BOOL
GET
Error := _Error OR _Overflow;
END_GET
END_PROPERTY

{attribute 'monitoring' := 'call'}
PROPERTY ErrorId : UDINT
GET
ErrorId := _ErrorId;
END_GET
END_PROPERTY

(* The parameter the loader stopped on, for diagnostics. *)
PROPERTY FailedParameterId : Tc3_Mc3Ptp.EAxisParameterId
GET
IF _Error AND (_Index >= 1) AND (_Index <= _Count) THEN
	FailedParameterId := _Bindings[_Index].ParameterId;
END_IF
END_GET
END_PROPERTY

METHOD Initialize
IF _Initialized OR _Error OR _Overflow THEN
	RETURN;
END_IF

IF NOT __ISVALIDREF(_Axis) THEN
	RETURN;
END_IF

// Nothing to read - trivially complete
IF _Count = 0 THEN
	_Initialized := TRUE;
	RETURN;
END_IF

// Wait for the NC axis to exist before asking it anything
IF _Axis.McToPlc.Std.AxisState = EAxisState.Invalid THEN
	RETURN;
END_IF

ReadParameter(Axis		  := _Axis,
			  Enable	  := TRUE,
			  ParameterId := _Bindings[_Index].ParameterId,
			  Mode		  := EReadMode.Once,
			  Valid		  =>,
			  Busy		  =>,
			  Error		  =>,
			  ErrorId	  =>,
			  Value		  => _Value);

IF ReadParameter.Error THEN
	_ErrorId := ReadParameter.ErrorId;
	_Error	 := TRUE;
	ReadParameter(Axis := _Axis, Enable := FALSE);
	RETURN;
END_IF

IF ReadParameter.Valid THEN
	_Bindings[_Index].Target^ := _Value;
	ReadParameter(Axis := _Axis, Enable := FALSE);

	IF _Index >= _Count THEN
		_Initialized := TRUE;
	ELSE
		_Index := _Index + 1;
	END_IF
END_IF
END_METHOD

{attribute 'monitoring' := 'call'}
PROPERTY Initialized : BOOL
GET
Initialized := _Initialized;
END_GET
SET
_Initialized := Initialized;

// Clearing the flag restarts the read from the first binding
IF NOT Initialized THEN
	_Index	 := 1;
	_Error	 := FALSE;
	_ErrorId := 0;
	ReadParameter(Axis := _Axis, Enable := FALSE);
END_IF
END_SET
END_PROPERTY

{attribute 'monitoring' := 'call'}
PROPERTY ParameterCount : UDINT
GET
ParameterCount := _Count;
END_GET
END_PROPERTY

END_FUNCTION_BLOCK

// ---- _Internal/Tracing/TcEventLogger.TcPOU
FUNCTION_BLOCK TcEventLogger IMPLEMENTS I_TraceLogger
VAR
	MessagesThisScan : DINT;
	Message			 : FB_TcMessage;
	Source			 : FB_TcSourceInfo;
	CurrentCycle	 : UDINT;
END_VAR

//FB_Init is always available implicitly and it is used primarily for initialization.

//The return value is not evaluated. For a specific influence, you can also declare the

//methods explicitly and provide additional code there with the standard initialization

//code. You can evaluate the return value.
METHOD FB_Init : BOOL
VAR_INPUT
	bInitRetains   : BOOL; // TRUE: the retain variables are initialized (reset warm / reset cold)
	bInCopyCode	   : BOOL; // TRUE: the instance will be copied to the copy code afterward (online change)   
	TracePublisher : I_TracePublisher;
END_VAR
IF ApplicationBaseParameter.EnableTcEventLogging THEN
	TracePublisher.Subscribe(THIS^);
END_IF
END_METHOD

METHOD LogMessage
VAR_INPUT
	Key		  : T_MaxString;
	Value	  : T_MaxString;
	SourceId  : UDINT := 0;
	TimeStamp : ULINT := 0;
	MessageId : UDINT := 1;
	Severity  : USINT := 1;
END_VAR
IF GETCURTASKINDEXEX() > 0 THEN
    IF TwinCAT_SystemInfoVarList._TaskInfo[GETCURTASKINDEXEX()].CycleCount <> CurrentCycle THEN
        CurrentCycle	 := TwinCAT_SystemInfoVarList._TaskInfo[GETCURTASKINDEXEX()].CycleCount;
        MessagesThisScan := 0;
    END_IF
    
    IF NOT (MessagesThisScan < TO_DINT(TwinCAT_SystemInfoVarList._TaskInfo[GETCURTASKINDEXEX()].CycleTime / 2000)) THEN
        RETURN;
    END_IF
END_IF
  
Source.sName := Key;
Source.nId	 := SourceId;
Message.Create(eventClass	:= TC_EVENT_CLASSES.Trace,
			   nEventId		:= MessageId,
			   eSeverity	:= USINT_To_TcEventSeverity(Severity),
			   ipSourceInfo := Source);

Message.ipArguments.Clear().AddString(Value);
Message.Send(TimeStamp);
Message.Release();
Source.Clear();
MessagesThisScan := MessagesThisScan + 1;
END_METHOD

END_FUNCTION_BLOCK

// ---- _Internal/Tracing/AdsLogger.TcPOU
FUNCTION_BLOCK AdsLogger IMPLEMENTS I_TraceLogger
VAR
	MessagesThisScan : DINT;
	CurrentCycle	 : UDINT;
END_VAR

//FB_Init is always available implicitly and it is used primarily for initialization.

//The return value is not evaluated. For a specific influence, you can also declare the

//methods explicitly and provide additional code there with the standard initialization

//code. You can evaluate the return value.
METHOD FB_Init : BOOL
VAR_INPUT
	bInitRetains   : BOOL; // TRUE: the retain variables are initialized (reset warm / reset cold)
	bInCopyCode	   : BOOL; // TRUE: the instance will be copied to the copy code afterward (online change)   
	TracePublisher : I_TracePublisher;
END_VAR
IF ApplicationBaseParameter.EnableAdsLogger THEN
	TracePublisher.Subscribe(THIS^);
END_IF
END_METHOD

METHOD LogMessage
VAR_INPUT
	Key		  : T_MaxString;
	Value	  : T_MaxString;
	SourceId  : UDINT := 0;
	TimeStamp : ULINT := 0;
	MessageId : UDINT := 1;
	Severity  : USINT := 1;
END_VAR
IF GETCURTASKINDEXEX() > 0 THEN
    IF TwinCAT_SystemInfoVarList._TaskInfo[GETCURTASKINDEXEX()].CycleCount <> CurrentCycle THEN
        CurrentCycle	 := TwinCAT_SystemInfoVarList._TaskInfo[GETCURTASKINDEXEX()].CycleCount;
        MessagesThisScan := 0;
    END_IF
    
    IF NOT (MessagesThisScan < TO_DINT(TwinCAT_SystemInfoVarList._TaskInfo[GETCURTASKINDEXEX()].CycleTime / 2000)) THEN
        RETURN;
    END_IF
END_IF


CASE Severity OF
	0, 1:
		ADSLOGSTR(ADSLOG_MSGTYPE_LOG OR ADSLOG_MSGTYPE_HINT, Concat(Value, ': %s'), Key);

	2:
		ADSLOGSTR(ADSLOG_MSGTYPE_LOG OR ADSLOG_MSGTYPE_WARN, Concat(Value, ': %s'), Key);

	3, 4:
		ADSLOGSTR(ADSLOG_MSGTYPE_LOG OR ADSLOG_MSGTYPE_ERROR, Concat(Value, ': %s'), Key);
END_CASE

MessagesThisScan := MessagesThisScan + 1;
END_METHOD

END_FUNCTION_BLOCK

// ---- Components/ADS/AdsReadWrite.TcPOU
FUNCTION_BLOCK AdsReadWrite EXTENDS CyclicComponent IMPLEMENTS I_AdsRW
VAR
	{attribute 'hide'}
	_AmsNetId : T_AmsNetId;
	{attribute 'hide'}
	_AmsPort : T_AmsPort;
	{attribute 'hide'}
	_AdsComMode		  : E_AdsComMode := eAdsComModeSecureCom;
	AdsRead			  : ADSREAD;
	AdsWrite		  : ADSWRITE;
	ReadAdsSymByName  : FB_ReadAdsSymByName;
	WriteAdsSymByName : FB_WriteAdsSymByName;
END_VAR

PROPERTY AdsComMode : E_AdsComMode
SET
_AdsComMode := AdsComMode;
END_SET
END_PROPERTY

{attribute 'monitoring' := 'call'}
PROPERTY AmsNetId : T_AmsNetId
GET
AmsNetId := _AmsNetId;
END_GET
SET
_AmsNetId := AmsNetId;
END_SET
END_PROPERTY

{attribute 'monitoring' := 'call'}
PROPERTY AmsPort : T_AmsPort
GET
AmsPort := _AmsPort;
END_GET
SET
_AmsPort := AmsPort;
END_SET
END_PROPERTY

{attribute 'monitoring' := 'call'}
PROPERTY Busy : BOOL
GET
Busy := AdsWrite.BUSY OR AdsRead.BUSY OR ReadAdsSymByName.bBusy OR WriteAdsSymByName.bBusy;
END_GET
END_PROPERTY

METHOD CyclicLogic
AdsRead(NETID := _AmsNetId, PORT := _AmsPort, TMOUT := DEFAULT_ADS_TIMEOUT);
AdsRead.READ := FALSE;
AdsWrite(NETID := _AmsNetId, PORT := _AmsPort, TMOUT := DEFAULT_ADS_TIMEOUT);
AdsWrite.WRITE := FALSE;

//
ReadAdsSymByName(sNetId		   := _AmsNetId,
				 nPort		   := _AmsPort,
				 tTimeout	   := DEFAULT_ADS_TIMEOUT,
				 eComMode	   := _AdsComMode,
				 bClearOnError := TRUE);

ReadAdsSymByName.bRead := FALSE;

//
WriteAdsSymByName(sNetId   := _AmsNetId,
				  nPort	   := _AmsPort,
				  tTimeout := DEFAULT_ADS_TIMEOUT,
				  eComMode := _AdsComMode);

WriteAdsSymByName.bWrite := FALSE;
END_METHOD

{attribute 'monitoring' := 'call'}
PROPERTY Error : BOOL
GET
Error := AdsWrite.ERR OR AdsRead.ERR OR ReadAdsSymByName.bError OR WriteAdsSymByName.bError;
END_GET
END_PROPERTY

{attribute 'monitoring' := 'call'}
PROPERTY ErrorId : UDINT
GET
IF AdsWrite.ERR THEN
	ErrorID := AdsWrite.ERRID;
ELSIF AdsRead.ERR THEN
	ErrorID := AdsRead.ERRID;
ELSIF ReadAdsSymByName.bError THEN
	ErrorID := ReadAdsSymByName.nErrorId;
ELSIF WriteAdsSymByName.bError THEN
	ErrorID := WriteAdsSymByName.nErrorId;
ELSE
	ErrorID := 0;
END_IF
END_GET
END_PROPERTY

METHOD Read
VAR_INPUT
	IdxGrp	  : UDINT;
	IdxOffset : UDINT;
	pDestAddr : PVOID;
	Length	  : UDINT;
END_VAR
IF AdsRead.BUSY THEN
	RETURN;
END_IF

AdsRead.IDXGRP	 := IdxGrp;
AdsRead.IDXOFFS	 := IdxOffset;
AdsRead.LEN		 := Length;
AdsRead.DESTADDR := pDestAddr;
AdsRead.READ	 := TRUE;
END_METHOD

METHOD ReadBySymbol
VAR_INPUT
	SymbolName : STRING(255);
	pDestAddr  : PVOID;
	Length	   : UDINT;
END_VAR
IF ReadAdsSymByName.bBusy THEN
	RETURN;
END_IF

ReadAdsSymByName.sVarName  := SymbolName;
ReadAdsSymByName.nDestAddr := pDestAddr;
ReadAdsSymByName.nLen	   := Length;
ReadAdsSymByName.bRead	   := TRUE;
END_METHOD

METHOD Write
VAR_INPUT
	IdxGrp		: UDINT;
	IdxOffset	: UDINT;
	pSourceAddr : PVOID;
	Length		: UDINT;
END_VAR
IF AdsWrite.BUSY THEN
	RETURN;
END_IF

AdsWrite.IDXGRP	 := IdxGrp;
AdsWrite.IDXOFFS := IdxOffset;
AdsWrite.LEN	 := Length;
AdsWrite.SRCADDR := pSourceAddr;
AdsWrite.WRITE	 := TRUE;
END_METHOD

METHOD WriteBySymbol
VAR_INPUT
	SymbolName	: STRING(255);
	pSourceAddr : PVOID;
	Length		: UDINT;
END_VAR
IF WriteAdsSymByName.bBusy THEN
	RETURN;
END_IF

WriteAdsSymByName.sVarName := SymbolName;
WriteAdsSymByName.nSrcAddr := pSourceAddr;
WriteAdsSymByName.nLen	   := Length;
WriteAdsSymByName.bWrite   := TRUE;
END_METHOD

END_FUNCTION_BLOCK

// ---- Components/Analog/AnalogInput.TcPOU
FUNCTION_BLOCK AnalogInput EXTENDS Component IMPLEMENTS I_AnalogInput, I_AnalogScalable, I_CalibratableLinear
VAR
	Input			 : REFERENCE TO INT;
	Forcible		 : ForcibleInt(_Name);
	_Scale			 : I_AnalogScale;
	_CalibrateLinear : I_CalibrateLinear;
	_CalibrateCustom : I_TransformLRealValue;
END_VAR

VAR
	{attribute 'hide'}
	DefaultScale : AnalogScale;
	{attribute 'hide'}
	DefaultCalibration : Calibrate;
END_VAR

PROPERTY CalibrateCustom : I_TransformLrealValue
SET
_CalibrateCustom := CalibrateCustom;
END_SET
END_PROPERTY

PROPERTY CalibrateLinear : I_CalibrateLinear
GET
CalibrateLinear := _CalibrateLinear;
END_GET
SET
_CalibrateLinear := CalibrateLinear;
END_SET
END_PROPERTY

(*FB_Init is always available implicitly and it is used primarily for initialization.
The return value is not evaluated. For a specific influence, you can also declare the
methods explicitly and provide additional code there with the standard initialization
code. You can evaluate the return value.*)
METHOD FB_Init : BOOL
VAR_INPUT
	(* TRUE: the retain variables are initialized (reset warm / reset cold)*)
	bInitRetains : BOOL;

	(* TRUE: the instance will be copied to the copy code afterward (online change)   *)
	bInCopyCode : BOOL;
	Name		: T_MaxString;
	Input		: REFERENCE TO INT;
END_VAR
_Scale			 := DefaultScale;
_CalibrateLinear := DefaultCalibration;
THIS^.Input		 REF= Input;
END_METHOD

{attribute 'monitoring' := 'call'}
PROPERTY Force : E_ForceState
GET
Force := Forcible.CurrentForceState;
END_GET
SET
VAR
	ForceString : T_MaxString := TO_STRING(Force);
END_VAR
Forcible.SetForceState(Force);
END_SET
END_PROPERTY

PROPERTY ForceValue : INT
GET
ForceValue := Forcible.ForceValue;
END_GET
SET
Forcible.ForceValue := ForceValue;
END_SET
END_PROPERTY

{attribute 'monitoring' := 'call'}
PROPERTY RawValue : INT
GET
Forcible.Input := Input;
RawValue	   := Forcible.Output;
END_GET
END_PROPERTY

PROPERTY Scale : I_AnalogScale
GET
Scale := _Scale;
END_GET
SET
_Scale := Scale;
END_SET
END_PROPERTY

{attribute 'monitoring' := 'call'}
PROPERTY Value : LREAL
GET
IF _CalibrateCustom = 0 THEN
	Value := _CalibrateLinear.Transform(_Scale.Transform(RawValue));
ELSE
	Value := _CalibrateCustom.Transform(_Scale.Transform(RawValue));
END_IF
END_GET
END_PROPERTY

END_FUNCTION_BLOCK

// ---- Utilities/Force/ForcibleInt.TcPOU
FUNCTION_BLOCK ForcibleInt
VAR
	Name			   : T_MaxString;
	_CurrentForceState : E_ForceState;
	ForceEvent		   : FB_TcAlarm;
	RequestedValue	   : INT;
	_Output			   : INT;
	_ForceValue : INT;
END_VAR

{attribute 'monitoring' := 'call'}
PROPERTY CurrentForceState : E_ForceState
GET
CurrentForceState := _CurrentForceState;
END_GET
END_PROPERTY

//FB_Init is always available implicitly and it is used primarily for initialization.

//The return value is not evaluated. For a specific influence, you can also declare the

//methods explicitly and provide additional code there with the standard initialization

//code. You can evaluate the return value.
METHOD FB_Init : BOOL
VAR_INPUT
	bInitRetains : BOOL; // TRUE: the retain variables are initialized (reset warm / reset cold)
	bInCopyCode	 : BOOL; // TRUE: the instance will be copied to the copy code afterward (online change) 
	Name		 : T_MaxString;
END_VAR
THIS^.Name := Name;
{analysis -15}
IF NOT ForceEvent.EqualsToEventEntryEx(TC_EVENTS.IO.ForceActive) THEN
	ForceEvent.CreateEx(TC_EVENTS.IO.ForceActive, 0);
END_IF
END_METHOD

PROPERTY ForceValue : INT
GET
ForceValue := _ForceValue;
END_GET
SET
_ForceValue := ForceValue;
END_SET
END_PROPERTY

{attribute 'monitoring' := 'call'}
PROPERTY Input : INT
SET
RequestedValue := Input;
ResolveOutput();
END_SET
END_PROPERTY

{attribute 'monitoring' := 'call'}
PROPERTY Output : INT
GET
Output := _Output;
END_GET
END_PROPERTY

METHOD PRIVATE ResolveOutput
VAR
	ForceString : T_MaxString := TO_STRING(_CurrentForceState);
END_VAR
CASE _CurrentForceState OF
	E_ForceState.Unforced:
		_Output := RequestedValue;
		ForceEvent.Clear();

	E_ForceState.ForceOn:
		IF NOT ForceEvent.bActive THEN
			ForceEvent.ipArguments.Clear().AddString(Name).AddString(ForceString);
			ForceEvent.Raise();
		END_IF

		_Output := _ForceValue;

	E_ForceState.ForceOff:
		IF NOT ForceEvent.bActive THEN
			ForceEvent.ipArguments.Clear().AddString(Name).AddString(ForceString);
			ForceEvent.Raise();
		END_IF

		_Output := 0;
END_CASE
END_METHOD

METHOD SetForceState
VAR_INPUT
	ForceState : E_ForceState;
END_VAR
IF ForceState = _CurrentForceState THEN
	RETURN;
END_IF

_CurrentForceState := ForceState;
ResolveOutput();
END_METHOD

END_FUNCTION_BLOCK

// ---- Utilities/Scaling/AnalogScale.TcPOU
FUNCTION_BLOCK AnalogScale IMPLEMENTS I_AnalogScale
VAR
	_InputMinimum  : LREAL := -32768;
	_InputMaximum  : LREAL := 32767;
	_OutputMinimum : LREAL := -32768;
	_OutputMaximum : LREAL := 32767;
END_VAR

PROPERTY InputMaximum : LREAL
GET
InputMaximum := _InputMaximum;
END_GET
SET
_InputMaximum := InputMaximum;
END_SET
END_PROPERTY

PROPERTY InputMinimum : LREAL
GET
InputMinimum := _InputMinimum;
END_GET
SET
_InputMinimum := InputMinimum;
END_SET
END_PROPERTY

PROPERTY OutputMaximum : LREAL
GET
OutputMaximum := _OutputMaximum;
END_GET
SET
_OutputMaximum := OutputMaximum;
END_SET
END_PROPERTY

PROPERTY OutputMinimum : LREAL
GET
OutputMinimum := _OutputMinimum;
END_GET
SET
_OutputMinimum := OutputMinimum;
END_SET
END_PROPERTY

METHOD Transform : LREAL
VAR_INPUT
	Value	: LREAL;
	Reverse : BOOL := FALSE;
END_VAR

VAR_INST
	Slope : LREAL;
END_VAR
//Scale is invalid
IF _InputMinimum >= _InputMaximum THEN
	Transform := 0;
	RETURN;
ELSIF _OutputMinimum >= _OutputMaximum THEN
	Transform := 0;
	RETURN;
END_IF

//Input is invalid
IF Value <= _InputMinimum THEN
	Transform := _OutputMinimum;
	RETURN;
ELSIF Value >= _InputMaximum THEN
	Transform := _OutputMaximum;
	RETURN;
END_IF

//I/O ok--scale it
IF (_InputMaximum - _InputMinimum) <> 0.0 THEN
	Slope := (_OutputMaximum - _OutputMinimum) / (_InputMaximum - _InputMinimum);
ELSE
	Slope := 0.0;
END_IF

Transform := Slope * (Value - _InputMinimum) + _OutputMinimum;
END_METHOD

END_FUNCTION_BLOCK

// ---- Utilities/Scaling/Calibrate.TcPOU
FUNCTION_BLOCK Calibrate IMPLEMENTS I_CalibrateLinear
VAR
	_Gain	: LREAL := 1;
	_Offset : LREAL := 0;
END_VAR

PROPERTY Gain : LREAL
SET
_Gain := Gain;
END_SET
END_PROPERTY

PROPERTY Offset : LREAL
SET
_Offset := Offset;
END_SET
END_PROPERTY

METHOD Transform : LREAL
VAR_INPUT
	Value	: LREAL;
	Reverse : BOOL := FALSE;
END_VAR
IF Reverse THEN
	Transform := (Value - _Offset) / _Gain;
ELSE
	Transform := Value * _Gain + _Offset;
END_IF
END_METHOD

END_FUNCTION_BLOCK

// ---- Components/Analog/AnalogInput_Generic.TcPOU
FUNCTION_BLOCK AnalogInput_Generic EXTENDS AnalogInput IMPLEMENTS I_AnalogChannel_Generic
VAR
	Status : REFERENCE TO ST_AnalogInputStatus_Generic;
END_VAR

PROPERTY DataValid : BOOL
GET
DataValid := NOT Status.WcState;
END_GET
END_PROPERTY

PROPERTY Error : BOOL
GET
Error := Status.Error;
END_GET
END_PROPERTY

(*FB_Init is always available implicitly and it is used primarily for initialization.
The return value is not evaluated. For a specific influence, you can also declare the
methods explicitly and provide additional code there with the standard initialization
code. You can evaluate the return value.*)
METHOD FB_Init : BOOL
VAR_INPUT
	(* TRUE: the retain variables are initialized (reset warm / reset cold)*)
	bInitRetains : BOOL;

	(* TRUE: the instance will be copied to the copy code afterward (online change)   *)
	bInCopyCode : BOOL;
	Name		: T_MaxString;
	Input		: REFERENCE TO INT;
	Status		: REFERENCE TO ST_AnalogInputStatus_Generic;
END_VAR
THIS^.Status REF= Status;
END_METHOD

PROPERTY Overrange : BOOL
GET
Overrange := Status.Overrange;
END_GET
END_PROPERTY

PROPERTY Underrange : BOOL
GET
Underrange := Status.Underrrange;
END_GET
END_PROPERTY

END_FUNCTION_BLOCK

// ---- Components/Analog/AnalogInput_Standard.TcPOU
FUNCTION_BLOCK AnalogInput_Standard EXTENDS AnalogInput IMPLEMENTS I_AnalogChannel_Standard
VAR
	Status : REFERENCE TO ST_AnalogInputStatus_EL30xx;
END_VAR

PROPERTY DataValid : BOOL
GET
DataValid := NOT Status.TxPDOState;
END_GET
END_PROPERTY

PROPERTY Error : BOOL
GET
Error := Status.Error;
END_GET
END_PROPERTY

(*FB_Init is always available implicitly and it is used primarily for initialization.
The return value is not evaluated. For a specific influence, you can also declare the
methods explicitly and provide additional code there with the standard initialization
code. You can evaluate the return value.*)
METHOD FB_Init : BOOL
VAR_INPUT
	(* TRUE: the retain variables are initialized (reset warm / reset cold)*)
	bInitRetains : BOOL;

	(* TRUE: the instance will be copied to the copy code afterward (online change)   *)
	bInCopyCode : BOOL;
	Name		: T_MaxString;
	Input		: REFERENCE TO INT;
	Status		: REFERENCE TO ST_AnalogInputStatus_EL30xx;
END_VAR
THIS^.Status REF= Status;
END_METHOD

PROPERTY Limit1High : BOOL
GET
Limit1High := Status.Limit1H;
END_GET
END_PROPERTY

PROPERTY Limit1Low : BOOL
GET
Limit1Low := Status.Limit1L;
END_GET
END_PROPERTY

PROPERTY Limit2High : BOOL
GET
Limit2High := Status.Limit2H;
END_GET
END_PROPERTY

PROPERTY Limit2Low : BOOL
GET
Limit2Low := Status.Limit2L;
END_GET
END_PROPERTY

PROPERTY Overrange : BOOL
GET
Overrange := Status.Overrange;
END_GET
END_PROPERTY

PROPERTY Underrange : BOOL
GET
Underrange := Status.Underrrange;
END_GET
END_PROPERTY

END_FUNCTION_BLOCK

// ---- Components/Analog/AnalogOutput.TcPOU
FUNCTION_BLOCK AnalogOutput EXTENDS Component IMPLEMENTS I_AnalogOutput, I_AnalogScalable, I_CalibratableLinear
VAR
	Output			 : REFERENCE TO INT;
	Forcible		 : ForcibleInt(_Name);
	_Scale			 : I_AnalogScale;
	_CalibrateLinear : I_CalibrateLinear;
	_CalibrateCustom : I_TransformLRealValue;
END_VAR

VAR
	{attribute 'hide'}
	DefaultScale : AnalogScale;
	{attribute 'hide'}
	DefaultCalibration : Calibrate;
END_VAR

PROPERTY CalibrateCustom : I_TransformLrealValue
SET
_CalibrateCustom := CalibrateCustom;
END_SET
END_PROPERTY

PROPERTY CalibrateLinear : I_CalibrateLinear
GET
CalibrateLinear := _CalibrateLinear;
END_GET
SET
_CalibrateLinear := CalibrateLinear;
END_SET
END_PROPERTY

(*FB_Init is always available implicitly and it is used primarily for initialization.
The return value is not evaluated. For a specific influence, you can also declare the
methods explicitly and provide additional code there with the standard initialization
code. You can evaluate the return value.*)
METHOD FB_Init : BOOL
VAR_INPUT
	(* TRUE: the retain variables are initialized (reset warm / reset cold)*)
	bInitRetains : BOOL;

	(* TRUE: the instance will be copied to the copy code afterward (online change)   *)
	bInCopyCode : BOOL;
	Name		: T_MaxString;
	Output		: REFERENCE TO INT;
END_VAR
_Scale			 := DefaultScale;
_CalibrateLinear := DefaultCalibration;
THIS^.Output	 REF= Output;
END_METHOD

{attribute 'monitoring' := 'call'}
PROPERTY Force : E_ForceState
GET
Force := Forcible.CurrentForceState;
END_GET
SET
VAR
	ForceString : T_MaxString := TO_STRING(Force);
END_VAR
Forcible.SetForceState(Force);
END_SET
END_PROPERTY

PROPERTY ForceValue : INT
GET
ForceValue := Forcible.ForceValue;
END_GET
SET
Forcible.ForceValue := ForceValue;
END_SET
END_PROPERTY

{attribute 'monitoring' := 'call'}
PROPERTY RawValue : INT
GET
RawValue := Output;
END_GET
SET
Forcible.Input := RawValue;
Output		   := Forcible.Output;
END_SET
END_PROPERTY

PROPERTY Scale : I_AnalogScale
GET
Scale := _Scale;
END_GET
SET
_Scale := Scale;
END_SET
END_PROPERTY

{attribute 'monitoring' := 'call'}
PROPERTY Value : LREAL
GET
IF _CalibrateCustom = 0 THEN
	Value := _CalibrateLinear.Transform(_Scale.Transform(RawValue));
ELSE
	Value := _CalibrateCustom.Transform(_Scale.Transform(RawValue));
END_IF
END_GET
SET
IF _CalibrateCustom = 0 THEN
	RawValue := LREAL_TO_INT(_Scale.Transform(_CalibrateLinear.Transform(Value, TRUE)));
ELSE
	RawValue := LREAL_TO_INT(_Scale.Transform(_CalibrateCustom.Transform(Value, TRUE)));
END_IF
END_SET
END_PROPERTY

END_FUNCTION_BLOCK

// ---- Components/Cylinder/Cylinder.TcPOU
FUNCTION_BLOCK Cylinder EXTENDS CyclicComponent IMPLEMENTS I_Cylinder
VAR
	ExtendOutput   : I_DigitalOutput;
	RetractOutput  : I_DigitalOutput;
	ExtendedInput  : I_DigitalInput;
	RetractedInput : I_DigitalInput;
	CylinderState  : E_CylinderState;
	{attribute 'hide'}
	_ExtendTimeout : TIME;
	{attribute 'hide'}
	_RetractTimeout : TIME;
	{attribute 'hide'}
	_Busy : BOOL;
	{attribute 'hide'}
	_Error : BOOL;
	{attribute 'hide'}
	_ErrorId : UDINT;
END_VAR

VAR
	{attribute 'hide'}
	NullEO : BOOL;
	{attribute 'hide'}
	NullExtendOutput : DigitalOutput('Null Digital Output', NullEO);
	{attribute 'hide'}
	NullRO : BOOL;
	{attribute 'hide'}
	NullRetractOutput : DigitalOutput('Null Digital Output', NullRO);
	{attribute 'hide'}
	NullEI : BOOL;
	{attribute 'hide'}
	NullExtendedInput : DigitalInput_NO('Null Digital Input', NullEI);
	{attribute 'hide'}
	NullRI : BOOL;
	{attribute 'hide'}
	NullRetractedInput : DigitalInput_NO('Null Digital Input', NullRI);
END_VAR

{attribute 'monitoring' := 'call'}
PROPERTY Busy : BOOL
GET
Busy := _Busy;
END_GET
END_PROPERTY

METHOD CyclicLogic
VAR_INST
	TON_RetractTimeout : TON;
	TON_ExtendTimeout  : TON;
END_VAR
NullEI := ExtendOutput.On;
NullRI := RetractOutput.On;
CASE CylinderState OF
	E_CylinderState.Undefined:
		IF ExtendedInput.IsActive THEN
			CylinderState := E_CylinderState.Extended;
		ELSIF RetractedInput.IsActive THEN
			CylinderState := E_CylinderState.Retracted;
		END_IF

	E_CylinderState.Extending:
		IF ExtendedInput.IsActive THEN
			CylinderState := E_CylinderState.Extended;
		END_IF

	E_CylinderState.Retracting:
		IF RetractedInput.IsActive THEN
			CylinderState := E_CylinderState.Retracted;
		END_IF
END_CASE

IF ExtendedInput.IsActive AND RetractedInput.IsActive THEN
	CylinderState := E_CylinderState.Undefined;
END_IF

// Generate Errors
IF CylinderState = E_CylinderState.Extending THEN
	IF _ExtendTimeout > T#0.0S THEN
		TON_ExtendTimeout(IN := TRUE, PT := _ExtendTimeout);
		IF TON_ExtendTimeout.Q THEN
			_Error	 := TRUE;
			_ErrorId := E_CylinderErrorId.ExtendTimeout;
		END_IF
	END_IF
ELSE
	TON_ExtendTimeout(IN := FALSE);
END_IF

IF CylinderState = E_CylinderState.Retracting THEN
	IF _RetractTimeout > T#0.0S THEN
		TON_RetractTimeout(IN := TRUE, PT := _RetractTimeout);
		IF TON_RetractTimeout.Q THEN
			_Error	 := TRUE;
			_ErrorId := E_CylinderErrorId.RetractTimeout;
		END_IF
	END_IF
ELSE
	TON_RetractTimeout(IN := FALSE);
END_IF

IF CylinderState = E_CylinderState.Extended THEN
	IF NOT ExtendedInput.IsActive THEN
		CylinderState := E_CylinderState.Undefined;
		_Error		  := TRUE;
		_ErrorId	  := E_CylinderErrorId.ExtendedPlausibility;
	END_IF
END_IF

IF CylinderState = E_CylinderState.Retracted THEN
	IF NOT RetractedInput.IsActive THEN
		CylinderState := E_CylinderState.Undefined;
		_Error		  := TRUE;
		_ErrorId	  := E_CylinderErrorId.RetractedPlausibility;
	END_IF
END_IF

IF ExtendedInput.IsActive AND RetractedInput.IsActive THEN
	CylinderState := E_CylinderState.Undefined;
	_Error		  := TRUE;
	_ErrorId	  := E_CylinderErrorId.BothSensorsActive;
END_IF

_Busy := (CylinderState = E_CylinderState.Extending) OR (CylinderState = E_CylinderState.Retracting);
END_METHOD

{attribute 'monitoring' := 'call'}
PROPERTY Error : BOOL
GET
Error := _Error;
END_GET
END_PROPERTY

{attribute 'monitoring' := 'call'}
PROPERTY ErrorId : UDINT
GET
ErrorID := _ErrorID;
END_GET
END_PROPERTY

METHOD Extend
IF CylinderState <> E_CylinderState.Extended THEN
	RetractOutput.On := FALSE;
	ExtendOutput.On	 := TRUE;
	CylinderState	 := E_CylinderState.Extending;
END_IF
END_METHOD

{attribute 'monitoring' := 'call'}
PROPERTY Extended : BOOL
GET
Extended := CylinderState = E_CylinderState.Extended;
END_GET
END_PROPERTY

{attribute 'monitoring' := 'call'}
PROPERTY Extending : BOOL
GET
Extending := CylinderState = E_CylinderState.Extending;
END_GET
END_PROPERTY

{attribute 'monitoring' := 'call'}
PROPERTY ExtendTimeout : TIME
GET
ExtendTimeout := _ExtendTimeout;
END_GET
SET
_ExtendTimeout := ExtendTimeout;
END_SET
END_PROPERTY

//FB_Init is always available implicitly and it is used primarily for initialization.

//The return value is not evaluated. For a specific influence, you can also declare the

//methods explicitly and provide additional code there with the standard initialization

//code. You can evaluate the return value.
METHOD FB_Init : BOOL
VAR_INPUT
	bInitRetains   : BOOL; // TRUE: the retain variables are initialized (reset warm / reset cold)
	bInCopyCode	   : BOOL; // TRUE: the instance will be copied to the copy code afterward (online change)  
	Name		   : T_MaxString;
	ExtendOutput   : I_DigitalOutput;
	RetractOutput  : I_DigitalOutput;
	ExtendedInput  : I_DigitalInput;
	RetractedInput : I_DigitalInput;
END_VAR
IF ExtendOutput = 0 THEN
	THIS^.ExtendOutput := NullExtendOutput;
ELSE
	THIS^.ExtendOutput := ExtendOutput;
END_IF

IF RetractOutput = 0 THEN
	THIS^.RetractOutput := NullRetractOutput;
ELSE
	THIS^.RetractOutput := RetractOutput;
END_IF

IF ExtendedInput = 0 THEN
	THIS^.ExtendedInput := NullExtendedInput;
ELSE
	THIS^.ExtendedInput := ExtendedInput;
END_IF

IF RetractedInput = 0 THEN
	THIS^.RetractedInput := NullRetractedInput;
ELSE
	THIS^.RetractedInput := RetractedInput;
END_IF
END_METHOD

METHOD Reset
_Error	 := FALSE;
_ErrorId := 0;
END_METHOD

METHOD Retract
IF CylinderState <> E_CylinderState.Retracted THEN
	ExtendOutput.On	 := FALSE;
	RetractOutput.On := TRUE;
	CylinderState	 := E_CylinderState.Retracting;
END_IF
END_METHOD

{attribute 'monitoring' := 'call'}
PROPERTY Retracted : BOOL
GET
Retracted := CylinderState = E_CylinderState.Retracted;
END_GET
END_PROPERTY

{attribute 'monitoring' := 'call'}
PROPERTY Retracting : BOOL
GET
Retracting := CylinderState = E_CylinderState.Retracting;
END_GET
END_PROPERTY

{attribute 'monitoring' := 'call'}
PROPERTY RetractTimeout : TIME
GET
RetractTimeout := _RetractTimeout;
END_GET
SET
_RetractTimeout := RetractTimeout;
END_SET
END_PROPERTY

END_FUNCTION_BLOCK

// ---- Components/Digital/DigitalOutput.TcPOU
FUNCTION_BLOCK DigitalOutput EXTENDS Component IMPLEMENTS I_DigitalOutput
VAR
	Output		   : REFERENCE TO BOOL;
	ForcableOutput : ForcibleBool(_Name);
END_VAR

//FB_Init is always available implicitly and it is used primarily for initialization.

//The return value is not evaluated. For a specific influence, you can also declare the

//methods explicitly and provide additional code there with the standard initialization

//code. You can evaluate the return value.
METHOD FB_Init : BOOL
VAR_INPUT
	bInitRetains : BOOL; // TRUE: the retain variables are initialized (reset warm / reset cold)
	bInCopyCode	 : BOOL; // TRUE: the instance will be copied to the copy code afterward (online change)   
	Name		 : T_MaxString;
	Output		 : REFERENCE TO BOOL;
END_VAR
THIS^.Output REF= Output;
END_METHOD

{attribute 'monitoring' := 'call'}
PROPERTY Force : E_ForceState
GET
Force := ForcableOutput.CurrentForceState;
END_GET
SET
ForcableOutput.SetForceState(Force);
Output := ForcableOutput.Output;
END_SET
END_PROPERTY

{attribute 'monitoring' := 'call'}
PROPERTY On : BOOL
GET
On := Output;
END_GET
SET
ForcableOutput.Input := On;
Output				 := ForcableOutput.Output;
END_SET
END_PROPERTY

END_FUNCTION_BLOCK

// ---- Utilities/Force/ForcibleBool.TcPOU
FUNCTION_BLOCK ForcibleBool
VAR
	Name			   : T_MaxString;
	_CurrentForceState : E_ForceState;
	ForceEvent		   : FB_TcAlarm;
	RequestedState	   : BOOL;
	_Output			   : BOOL;
END_VAR

{attribute 'monitoring' := 'call'}
PROPERTY CurrentForceState : E_ForceState
GET
CurrentForceState := _CurrentForceState;
END_GET
END_PROPERTY

//FB_Init is always available implicitly and it is used primarily for initialization.

//The return value is not evaluated. For a specific influence, you can also declare the

//methods explicitly and provide additional code there with the standard initialization

//code. You can evaluate the return value.
METHOD FB_Init : BOOL
VAR_INPUT
	bInitRetains : BOOL; // TRUE: the retain variables are initialized (reset warm / reset cold)
	bInCopyCode	 : BOOL; // TRUE: the instance will be copied to the copy code afterward (online change) 
	Name		 : T_MaxString;
END_VAR
THIS^.Name := Name;
{analysis -15}
IF NOT ForceEvent.EqualsToEventEntryEx(TC_EVENTS.IO.ForceActive) THEN
	ForceEvent.CreateEx(TC_EVENTS.IO.ForceActive, 0);
END_IF
END_METHOD

{attribute 'monitoring' := 'call'}
PROPERTY Input : BOOL
SET
RequestedState := Input;
ResolveOutput();
END_SET
END_PROPERTY

{attribute 'monitoring' := 'call'}
PROPERTY Output : BOOL
GET
Output := _Output;
END_GET
END_PROPERTY

METHOD PRIVATE ResolveOutput
VAR
	ForceString : T_MaxString := TO_STRING(_CurrentForceState);
END_VAR
CASE _CurrentForceState OF
	E_ForceState.Unforced:
		_Output := RequestedState;
		ForceEvent.Clear();

	E_ForceState.ForceOn:
		IF NOT ForceEvent.bActive THEN
			ForceEvent.ipArguments.Clear().AddString(Name).AddString(ForceString);
			ForceEvent.Raise();
		END_IF

		_Output := TRUE;

	E_ForceState.ForceOff:
		IF NOT ForceEvent.bActive THEN
			ForceEvent.ipArguments.Clear().AddString(Name).AddString(ForceString);
			ForceEvent.Raise();
		END_IF

		_Output := FALSE;
END_CASE
END_METHOD

METHOD SetForceState
VAR_INPUT
	ForceState : E_ForceState;
END_VAR
IF ForceState = _CurrentForceState THEN
	RETURN;
END_IF

_CurrentForceState := ForceState;
ResolveOutput();
END_METHOD

END_FUNCTION_BLOCK

// ---- Components/Digital/DigitalInput_NO.TcPOU
FUNCTION_BLOCK DigitalInput_NO EXTENDS Component IMPLEMENTS I_DigitalInput
VAR
	Input		  : REFERENCE TO BOOL;
	ForcibleInput : ForcibleBool(_Name);
END_VAR

//FB_Init is always available implicitly and it is used primarily for initialization.

//The return value is not evaluated. For a specific influence, you can also declare the

//methods explicitly and provide additional code there with the standard initialization

//code. You can evaluate the return value.
METHOD FB_Init : BOOL
VAR_INPUT
	bInitRetains : BOOL; // TRUE: the retain variables are initialized (reset warm / reset cold)
	bInCopyCode	 : BOOL; // TRUE: the instance will be copied to the copy code afterward (online change)   
	Name		 : T_MaxString;
	Input		 : REFERENCE TO BOOL;
END_VAR
THIS^.Input REF= Input;
END_METHOD

{attribute 'monitoring' := 'call'}
PROPERTY Force : E_ForceState
GET
Force := ForcibleInput.CurrentForceState;
END_GET
SET
VAR
	ForceString : T_MaxString := TO_STRING(Force);
END_VAR
ForcibleInput.SetForceState(Force);
END_SET
END_PROPERTY

{attribute 'monitoring' := 'call'}
PROPERTY IsActive : BOOL
GET
ForcibleInput.Input := Input;
IsActive			:= ForcibleInput.Output;
END_GET
END_PROPERTY

END_FUNCTION_BLOCK

// ---- Components/Cylinder/Cylinder_HMI.TcPOU
FUNCTION_BLOCK Cylinder_HMI EXTENDS HmiFunction
VAR
	Cylinder : I_Cylinder;
	{ attribute 'TcHmiSymbol.AddSymbol' }
	{ attribute 'TcHmiSymbol.AddSymbol.UserGroups' := '__SystemAdministrators,Admin' }
	Cylinder_HMI : ST_Cylinder_HMI;
END_VAR

PROPERTY ControlObject : I_Base
SET
__QueryInterface(ControlObject,Cylinder);
END_SET
END_PROPERTY

METHOD CyclicLogic
VAR_INST
	ExtendRT  : R_TRIG;
	RetractRT : R_TRIG;
END_VAR
IF Cylinder = 0 THEN
	RETURN;
END_IF

Cylinder_HMI.HmiEnabled := Enabled;
Cylinder_HMI.Name		:= Cylinder.Name;
Cylinder_HMI.Busy		:= Cylinder.Busy;
Cylinder_HMI.Error		:= Cylinder.Error;
Cylinder_HMI.ErrorId	:= Cylinder.ErrorId;
Cylinder_HMI.Extended	:= Cylinder.Extended;
Cylinder_HMI.Retracted	:= Cylinder.Retracted;
// HMI Commands
IF Enabled THEN
	ExtendRT(CLK := Cylinder_HMI.Extend.Active);
	IF ExtendRT.Q THEN
		IF Cylinder_HMI.Extend.Permissive.OK THEN
			Cylinder.Extend();
		END_IF
	END_IF

	RetractRT(CLK := Cylinder_HMI.Retract.Active);
	IF RetractRT.Q THEN
		IF Cylinder_HMI.Retract.Permissive.OK THEN
			Cylinder.Retract();
		END_IF
	END_IF
END_IF
END_METHOD

PROPERTY ExtendCommandName : STRING
GET
ExtendCommandName := Cylinder_HMI.Extend.Name;
END_GET
SET
Cylinder_HMI.Extend.Name := ExtendCommandName;
END_SET
END_PROPERTY

PROPERTY ExtendedName : STRING
GET
ExtendedName := Cylinder_HMI.ExtendedName;
END_GET
SET
Cylinder_HMI.ExtendedName := ExtendedName;
END_SET
END_PROPERTY

PROPERTY ExtendPermissive : I_Permissive
GET
ExtendPermissive := Cylinder_HMI.Extend.Permissive;
END_GET
END_PROPERTY

(*FB_Init is always available implicitly and it is used primarily for initialization.
The return value is not evaluated. For a specific influence, you can also declare the
methods explicitly and provide additional code there with the standard initialization
code. You can evaluate the return value.*)
METHOD FB_Init : BOOL
VAR_INPUT
	(* TRUE: the retain variables are initialized (reset warm / reset cold)*)
	bInitRetains : BOOL;

	(* TRUE: the instance will be copied to the copy code afterward (online change)   *)
	bInCopyCode : BOOL;
	Name		: T_MaxString;
	Cylinder	: I_Cylinder;
END_VAR
THIS^.Cylinder := Cylinder;
ControlType	   := 'Cylinder';
LinkObject	   := 'Cylinder_HMI';
END_METHOD

PROPERTY RetractCommandName : STRING
GET
RetractCommandName := Cylinder_HMI.Retract.Name;
END_GET
SET
Cylinder_HMI.Retract.Name := RetractCommandName;
END_SET
END_PROPERTY

PROPERTY RetractedName : STRING
GET
RetractedName := Cylinder_HMI.RetractedName;
END_GET
SET
Cylinder_HMI.RetractedName := RetractedName;
END_SET
END_PROPERTY

PROPERTY RetractPermissive : I_Permissive
GET
RetractPermissive := Cylinder_HMI.Retract.Permissive;
END_GET
END_PROPERTY

END_FUNCTION_BLOCK

// ---- HMI/HmiFunction.TcPOU
{attribute 'reflection'}
FUNCTION_BLOCK ABSTRACT HmiFunction EXTENDS CyclicComponent IMPLEMENTS I_HmiFunction
VAR
	{attribute 'instance-path'}
	{attribute 'noinit'}
	{attribute 'hide'}
	_InstancePath : STRING;
	{attribute 'hide'}
	_Enabled : BOOL := TRUE;
	{attribute 'hide'}
	_ControlType : STRING := 'Default';
	{attribute 'hide'}
	_LinkObject : STRING := 'DefaultFunction_HMI';
END_VAR

PROPERTY ABSTRACT ControlObject : I_Base
SET
END_SET
END_PROPERTY

{attribute 'monitoring' := 'call'}
PROPERTY ControlType : STRING
GET
ControlType := _ControlType;
END_GET
SET
_ControlType := ControlType;
END_SET
END_PROPERTY

METHOD CyclicLogic
END_METHOD

METHOD Disable
_Enabled := FALSE;
END_METHOD

METHOD Enable
_Enabled := TRUE;
END_METHOD

{attribute 'monitoring' := 'call'}
PROPERTY Enabled : BOOL
GET
Enabled := _Enabled;
END_GET
END_PROPERTY

{attribute 'monitoring' := 'call'}
PROPERTY InstancePath : STRING
GET
InstancePath := _InstancePath;
END_GET
END_PROPERTY

{attribute 'monitoring' := 'call'}
PROPERTY LinkObject : STRING
GET
LinkObject := _LinkObject;
END_GET
SET
_LinkObject := LinkObject;
END_SET
END_PROPERTY

END_FUNCTION_BLOCK

// ---- Components/Cylinder/Cylinder_TcEvents.TcPOU
FUNCTION_BLOCK Cylinder_TcEvents EXTENDS CyclicComponent IMPLEMENTS I_EventReactionTcEvents
VAR
	Cylinder : I_Cylinder;
	Events	 : TcEventClass(CONCAT(Name, ' Events'));
END_VAR

METHOD CyclicLogic
IF Cylinder.Error THEN
	CASE Cylinder.ErrorId OF
		E_CylinderErrorId.NoError:
			;

		E_CylinderErrorId.BothSensorsActive:
			Events.RaiseEvent(E_cylinder.BothSensorsActive);

		E_CylinderErrorId.ExtendedPlausibility:
			Events.RaiseEvent(E_cylinder.ExtendedPlausibility);

		E_CylinderErrorId.ExtendTimeout:
			Events.RaiseEvent(E_cylinder.ExtendTimeout);

		E_CylinderErrorId.RetractedPlausibility:
			Events.RaiseEvent(E_cylinder.RetractedPlausibility);

		E_CylinderErrorId.RetractTimeout:
			Events.RaiseEvent(E_cylinder.RetractTimeout);
	END_CASE
END_IF
END_METHOD

(*FB_Init is always available implicitly and it is used primarily for initialization.
The return value is not evaluated. For a specific influence, you can also declare the
methods explicitly and provide additional code there with the standard initialization
code. You can evaluate the return value.*)
METHOD FB_Init : BOOL
VAR_INPUT
	(* TRUE: the retain variables are initialized (reset warm / reset cold)*)
	bInitRetains : BOOL;

	(* TRUE: the instance will be copied to the copy code afterward (online change)   *)
	bInCopyCode : BOOL;
	Name		: T_MaxString;
	Cylinder	: I_Cylinder;
END_VAR
THIS^.Cylinder := Cylinder;
Events.GenerateTcEvents(Cylinder.Name, ADR(TC_events.Cylinder), SIZEOF(ST_Cylinder));
END_METHOD

METHOD GetHighestActiveEventReaction : DINT
GetHighestActiveEventReaction := Events.GetHighestActiveEventReaction();
END_METHOD

METHOD GetHighestActiveEventSeverity : TcEventSeverity
GetHighestActiveEventSeverity := Events.GetHighestActiveEventSeverity();
END_METHOD

METHOD Reset
Events.Reset();
END_METHOD

METHOD SetEventReactions
VAR_INPUT
	Verbose	 : DINT := 0;
	Info	 : DINT := 1;
	Warning	 : DINT := 2;
	Error	 : DINT := 3;
	Critical : DINT := 4;
END_VAR
Events.SetEventReactions(Verbose,
						 Info,
						 Warning,
						 Error,
						 Critical);
END_METHOD

END_FUNCTION_BLOCK

// ---- Events/TcEventClass.TcPOU
{attribute 'enable_dynamic_creation'}
FUNCTION_BLOCK TcEventClass EXTENDS CyclicComponent IMPLEMENTS I_EventClassTcEvents
VAR
	pEventClass				   : PVOID;
	pEventBuffer			   : POINTER TO PVOID;
	pEventTriggerBuffer		   : POINTER TO PVOID;
	pEventAutoResetBuffer	   : POINTER TO PVOID;
	NullEvent				   : FB_TcAlarm;
	NullBool				   : BOOL;
	NumberOfEvents			   : UDINT;
	HighestActiveEventSeverity : TcEventSeverity;
	EventReactionVerbose	   : DINT := 0;
	EventReactionInfo		   : DINT := 1;
	EventReactionWarning	   : DINT := 2;
	EventReactionError		   : DINT := 3;
	EventReactionCritical	   : DINT := 4;
	TcEventClassArguments	   : TcEventClassArguments;
END_VAR

METHOD PUBLIC Arguments : I_EventArguments
VAR_INPUT
	EventId : UDINT;
END_VAR

VAR
	pEvent : POINTER TO FB_TcAlarm;
END_VAR
IF CheckEventId(EventId) THEN
	pEvent := GetEventInstance(EventId);
	IF (pEvent <> 0) THEN
		TcEventClassArguments.Event := pEvent;
	ELSE
		TcEventClassArguments.Event := ADR(NullEvent);
	END_IF
ELSE
	TcEventClassArguments.Event := ADR(NullEvent);
END_IF

Arguments := TcEventClassArguments;
END_METHOD

METHOD PROTECTED CheckEventId : BOOL
VAR_INPUT
	EventId : UDINT;
END_VAR
CheckEventId := (EventID > 0) AND (EventId <= NumberOfEvents) AND (pEventBuffer <> 0);
END_METHOD

METHOD ClearEventById
VAR_INPUT
	EventId : UDINT;
END_VAR

VAR
	pEvent : POINTER TO FB_TcAlarm;
END_VAR
IF CheckEventId(EventId) THEN
	pEvent := GetEventInstance(EventId);
	IF (pEvent <> 0) THEN
		IF pEvent^.bRaised THEN
			pEvent^.Clear();
			FindActiveSeverity();
		END_IF
	END_IF
END_IF
END_METHOD

METHOD CyclicLogic
VAR
	i	   : UDINT;
	pEvent : POINTER TO FB_TcAlarm;
	pTrigger  : POINTER TO BOOL;
    AutoReset : BOOL;
END_VAR
FOR i := 1 TO NumberOfEvents DO
	pTrigger := GetEventTriggerInstance(i);
	IF (pTrigger <> 0) THEN
		pEvent	  := GetEventInstance(i);
		AutoReset := GetEventAutoResetInstance(i)^;
		IF (pEvent <> 0) AND_THEN AutoReset AND NOT pTrigger^ THEN
			pEvent^.Clear();
			FindActiveSeverity();
		END_IF

		IF (pEvent <> 0) AND_THEN pTrigger^ THEN
			pEvent^.Raise(0);
			FindActiveSeverity();
		END_IF
	END_IF
END_FOR
END_METHOD

METHOD Dispose
VAR
	i				: UDINT;
	pEvent			: POINTER TO FB_TcAlarm;
	pDispose		: POINTER TO TcEventClass;
	pEventAutoReset : POINTER TO BOOL;
END_VAR
pDispose := THIS;
FOR i := 1 TO NumberOfEvents DO
	pEvent := GetEventInstance(i);
	__DELETE(pEvent);
	pEventAutoReset := GetEventAutoResetInstance(i);
	__DELETE(pEventAutoReset);
END_FOR

__DELETE(pEventBuffer);
__DELETE(pDispose);
__DELETE(pEventTriggerBuffer);
__DELETE(pEventAutoResetBuffer);
END_METHOD

//FB_Exit must be implemented explicitly. If there is an implementation, then the

//method is called before the controller removes the code of the function block instance

//(implicit call). The return value is not evaluated.
METHOD FB_Exit : BOOL
VAR_INPUT
	bInCopyCode : BOOL; // TRUE: the exit method is called in order to leave the instance which will be copied afterwards (online change).  
END_VAR

VAR
	i				: UDINT;
	pEvent			: POINTER TO FB_TcAlarm;
	pEventAutoReset : POINTER TO BOOL;
END_VAR
FOR i := 1 TO NumberOfEvents DO
	pEvent := GetEventInstance(i);
	__DELETE(pEvent);
	pEventAutoReset := GetEventAutoResetInstance(i);
	__DELETE(pEventAutoReset);
END_FOR

__DELETE(pEventBuffer);
__DELETE(pEventTriggerBuffer);
__DELETE(pEventAutoResetBuffer);
END_METHOD

METHOD PROTECTED FindActiveSeverity
VAR
	i	   : UDINT;
	pEvent : POINTER TO FB_TcAlarm;
END_VAR
HighestActiveEventSeverity := Global.TcEventSeverity.Verbose;
FOR i := 1 TO NumberOfEvents DO
	pEvent := GetEventInstance(i);
	IF (pEvent <> 0) AND_THEN pEvent^.bRaised AND_THEN pEvent^.eSeverity > HighestActiveEventSeverity THEN
		HighestActiveEventSeverity := pEvent^.eSeverity;
	END_IF
END_FOR
END_METHOD

METHOD PUBLIC GenerateTcEvents
VAR_INPUT
	Name   : T_MaxString;
	pClass : PVOID; // ADR(TC_Events.XY) - TC Event Class in TypeSystem
	nSize  : UDINT; // SIZEOF(ST_XY) - TC Event Class in TypeSystem
END_VAR

VAR
	i				 : UDINT;
	pEventDef		 : POINTER TO TcEventEntry;
	pEvent			 : POINTER TO FB_TcAlarm;
	pBuffer			 : PVOID;
	ppBuffer		 : POINTER TO POINTER TO FB_TcAlarm;
	SourceInfo		 : FB_TcSourceInfo;
	pEventAutoReset	 : POINTER TO BOOL;
	ppEventAutoReset : POINTER TO POINTER TO BOOL;
END_VAR
NumberOfEvents		  := nSize / SIZEOF(TcEventEntry);
pEventBuffer		  := __NEW(PVOID, NumberOfEvents);
pEventTriggerBuffer	  := __NEW(PVOID, NumberOfEvents);
pEventAutoResetBuffer := __NEW(PVOID, NumberOfEvents);
pEventClass			  := pClass;
IF pEventBuffer <> 0 THEN
	SourceInfo.ResetToDefault();
	SourceInfo.sName := Name;
	FOR i := 1 TO NumberOfEvents DO
		pEvent	  := __NEW(FB_TcAlarm);
		ppBuffer  := pEventBuffer + ((i - 1) * SIZEOF(PVOID));
		ppBuffer^ := pEvent;
		pEventDef := pEventClass + ((i - 1) * SIZEOF(TcEventEntry));
		pEvent^.CreateEx2(pEventDef^, SourceInfo);

		//
		pEventAutoReset	  := __NEW(BOOL);
		ppEventAutoReset  := pEventAutoResetBuffer + ((i - 1) * SIZEOF(PVOID));
		ppEventAutoReset^ := pEventAutoReset;
	END_FOR
END_IF
END_METHOD

METHOD PROTECTED GetEventAutoResetInstance : POINTER TO BOOL
VAR_INPUT
	EventId : UDINT;
END_VAR

VAR
	ppEventAutoReset : POINTER TO POINTER TO BOOL;
END_VAR
IF CheckEventId(EventId) THEN
	ppEventAutoReset := pEventAutoResetBuffer + ((EventId - 1) * SIZEOF(PVOID));
	GetEventAutoResetInstance := ppEventAutoReset^;
ELSE
	GetEventAutoResetInstance := ADR(NullBool);
END_IF
END_METHOD

METHOD PROTECTED GetEventInstance : POINTER TO FB_TcAlarm
VAR_INPUT
	EventId : UDINT;
END_VAR

VAR
	ppEvent : POINTER TO POINTER TO FB_TcAlarm;
END_VAR
IF CheckEventId(EventId) THEN
	ppEvent			 := pEventBuffer + ((EventId - 1) * SIZEOF(PVOID));
	GetEventInstance := ppEvent^;
ELSE
	GetEventInstance := ADR(NullEvent);
END_IF
END_METHOD

METHOD PROTECTED GetEventTriggerInstance : POINTER TO BOOL
VAR_INPUT
	EventId : UDINT;
END_VAR

VAR
	ppEventTrigger : POINTER TO POINTER TO BOOL;
END_VAR
IF CheckEventId(EventId) THEN
	ppEventTrigger := pEventTriggerBuffer + ((EventId - 1) * SIZEOF(PVOID));
	GetEventTriggerInstance := ppEventTrigger^;
ELSE
	GetEventTriggerInstance := ADR(NullBool);
END_IF
END_METHOD

METHOD GetHighestActiveEventReaction : DINT
CASE HighestActiveEventSeverity OF
	TcEventSeverity.Verbose:
		GetHighestActiveEventReaction := EventReactionVerbose;

	TcEventSeverity.Info:
		GetHighestActiveEventReaction := EventReactionInfo;

	TcEventSeverity.Warning:
		GetHighestActiveEventReaction := EventReactionWarning;

	TcEventSeverity.Error:
		GetHighestActiveEventReaction := EventReactionError;

	TcEventSeverity.Critical:
		GetHighestActiveEventReaction := EventReactionCritical;
END_CASE
END_METHOD

METHOD GetHighestActiveEventSeverity : TcEventSeverity
GetHighestActiveEventSeverity := HighestActiveEventSeverity;
END_METHOD

{attribute 'monitoring' := 'call'}
PROPERTY IsResettable : BOOL
GET
VAR
	i		  : UDINT;
	pEvent	  : POINTER TO FB_TcAlarm;
	pTrigger  : POINTER TO BOOL;
END_VAR
IsResettable := FALSE;
FOR i := 1 TO NumberOfEvents DO
	pTrigger := GetEventTriggerInstance(i);
	IF (pTrigger <> 0) THEN
		pEvent := GetEventInstance(i);
		IF (pEvent <> 0) AND_THEN NOT pTrigger^ AND pEvent^.bRaised THEN
			IsResettable := TRUE;
		END_IF
	END_IF
END_FOR
END_GET
END_PROPERTY

METHOD RaiseEvent
VAR_INPUT
	EventId	  : UDINT;
END_VAR

VAR
	pEvent : POINTER TO FB_TcAlarm;
END_VAR
IF CheckEventId(EventId) THEN
	pEvent := GetEventInstance(EventId);
	IF (pEvent <> 0) THEN
		IF NOT pEvent^.bRaised THEN
			pEvent^.Raise();
			IF pEvent^.eSeverity > HighestActiveEventSeverity THEN
				HighestActiveEventSeverity := pEvent^.eSeverity;
			END_IF

			pEvent^.ipArguments.Clear();
		END_IF
	END_IF
END_IF
END_METHOD

METHOD Reset
VAR
	i		 : UDINT;
	pEvent	 : POINTER TO FB_TcAlarm;
	pTrigger : POINTER TO BOOL;
END_VAR
FOR i := 1 TO NumberOfEvents DO
	pTrigger := GetEventTriggerInstance(i);
	pEvent	 := GetEventInstance(i);
	IF (pEvent <> 0) THEN
		IF (pTrigger <> 0) AND_THEN NOT pTrigger^ THEN
			pEvent^.Clear();
		END_IF

		IF (pTrigger = 0) THEN
			pEvent^.Clear();
		END_IF
	END_IF
END_FOR

HighestActiveEventSeverity := Global.TcEventSeverity.Verbose;
END_METHOD

METHOD ResetBySeverity : BOOL
VAR_INPUT
	Severity : UDINT;
END_VAR

VAR
	i	   : UDINT;
	pEvent : POINTER TO FB_TcAlarm;
END_VAR
FOR i := 1 TO NumberOfEvents DO
	pEvent := GetEventInstance(i);
	IF (pEvent <> 0) AND_THEN (pEvent^.eSeverity <= TO_DINT(Severity)) THEN
		pEvent^.Clear();
	END_IF
END_FOR

FindActiveSeverity();
ResetBySeverity := TRUE;
END_METHOD

METHOD SetEvent
VAR_INPUT
	EventId	  : UDINT;
	Trigger	  : POINTER TO BOOL;
	AutoReset : BOOL;
END_VAR

VAR
	pBool : POINTER TO BOOL;
END_VAR
IF CheckEventId(EventId) THEN
	IF Trigger <> 0 THEN
		SetEventTriggerInstance(EventId, Trigger);
	END_IF

	pBool  := GetEventAutoResetInstance(EventId);
	pBool^ := AutoReset;
END_IF
END_METHOD

METHOD SetEventReactions
VAR_INPUT
	Verbose	 : DINT := 0;
	Info	 : DINT := 1;
	Warning	 : DINT := 2;
	Error	 : DINT := 3;
	Critical : DINT := 4;
END_VAR
EventReactionVerbose  := Verbose;
EventReactionInfo	  := Info;
EventReactionWarning  := Warning;
EventReactionError	  := Error;
EventReactionCritical := Critical;
END_METHOD

METHOD PROTECTED SetEventTriggerInstance
VAR_INPUT
	EventId : UDINT;
    Trigger : POINTER TO BOOL;
END_VAR

VAR
	ppEventTrigger : POINTER TO POINTER TO BOOL;
END_VAR
IF CheckEventId(EventId) THEN
	ppEventTrigger	:= pEventTriggerBuffer + ((EventId - 1) * SIZEOF(PVOID));
	ppEventTrigger^ := Trigger;
END_IF
END_METHOD

END_FUNCTION_BLOCK

// ---- _Internal/Events/TcEventClassArguments.TcPOU
FUNCTION_BLOCK TcEventClassArguments IMPLEMENTS I_EventArguments
VAR
	pArgumentEvent : POINTER TO FB_TcAlarm;
END_VAR

METHOD AddString : I_EventArguments
VAR_INPUT
	Argument : STRING;
END_VAR
IF pArgumentEvent <> 0 THEN
	pArgumentEvent^.ipArguments.AddString(Argument);
END_IF

AddString := THIS^;
END_METHOD

